// ---- VISUs/EtherCAT_Diag2.TcVIS
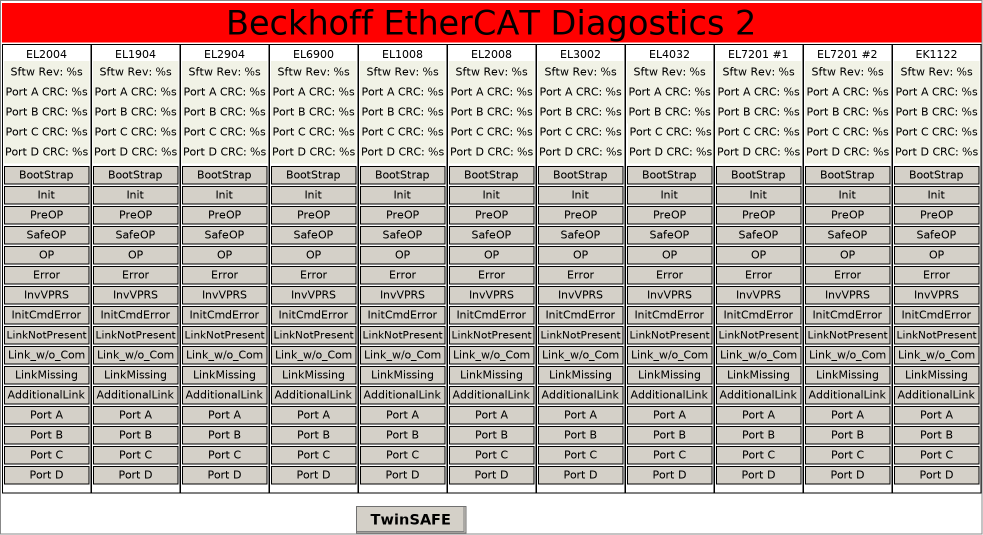
VISUALIZATION EtherCAT_Diag2  // 983x535
    Button (356,506 110x27), "TwinSAFE"
        OnMouseClick: change screen: TwinSAFE
    RoundedRectangle (2,3 979x39), "Beckhoff EtherCAT Diagostics 2"
    Group (2,42 89x451)
        RoundedRectangle (0,2 89x449)
        Label (2,0 85x25), "EL2004"
        Rectangle (2,19 85x22), "Sftw Rev: %s", text variable: g_iHMI_ProdCodeEL2004
        Rectangle (2,39 85x22), "Port A CRC: %s", text variable: g_stHMI_EL2004CrcErrorEx.portA
        Rectangle (2,59 85x22), "Port B CRC: %s", text variable: g_stHMI_EL2004CrcErrorEx.portB
        Rectangle (2,79 85x22), "Port C CRC: %s", text variable: g_stHMI_EL2004CrcErrorEx.portC
        Rectangle (2,99 85x22), "Port D CRC: %s", text variable: g_stHMI_EL2004CrcErrorEx.portD
        Rectangle (2,124 85x18), "BootStrap", colour toggle: g_stHMI_EL2004EcSlaveStateBits.bBootStrap
        Rectangle (2,144 85x18), "Init", colour toggle: g_stHMI_EL2004EcSlaveStateBits.bInit
        Rectangle (2,164 85x18), "PreOP", colour toggle: g_stHMI_EL2004EcSlaveStateBits.bPreop
        Rectangle (2,184 85x18), "SafeOP", colour toggle: g_stHMI_EL2004EcSlaveStateBits.bSafeOp
        Rectangle (2,204 85x18), "OP", colour toggle: g_stHMI_EL2004EcSlaveStateBits.bOp
        Rectangle (2,224 85x18), "Error", colour toggle: g_stHMI_EL2004EcSlaveStateBits.bError
        Rectangle (2,244 85x18), "InvVPRS", colour toggle: g_stHMI_EL2004EcSlaveStateBits.bInvVPRS
        Rectangle (2,264 85x18), "InitCmdError", colour toggle: g_stHMI_EL2004EcSlaveStateBits.bInitCmdError
        Rectangle (2,284 85x18), "LinkNotPresent", colour toggle: g_stHMI_EL2004EcSlaveStateBits.bLinkNotPresent
        Rectangle (2,304 85x18), "Link_w/o_Com", colour toggle: g_stHMI_EL2004EcSlaveStateBits.bLinkWithoutComm
        Rectangle (2,324 85x18), "LinkMissing", colour toggle: g_stHMI_EL2004EcSlaveStateBits.bLinkMissing
        Rectangle (2,344 85x18), "AdditionalLink", colour toggle: g_stHMI_EL2004EcSlaveStateBits.bAdditionalLink
        Rectangle (2,364 85x18), "Port A", colour toggle: g_stHMI_EL2004EcSlaveStateBits.bPortA
        Rectangle (2,384 85x18), "Port B", colour toggle: g_stHMI_EL2004EcSlaveStateBits.bPortB
        Rectangle (2,404 85x18), "Port C", colour toggle: g_stHMI_EL2004EcSlaveStateBits.bPortC
        Rectangle (2,424 85x18), "Port D", colour toggle: g_stHMI_EL2004EcSlaveStateBits.bPortD
    Group (91,42 89x451)
        RoundedRectangle (0,2 89x449)
        Label (2,0 85x25), "EL1904"
        Rectangle (2,19 85x22), "Sftw Rev: %s", text variable: g_iHMI_ProdCodeEL1904
        Rectangle (2,39 85x22), "Port A CRC: %s", text variable: g_stHMI_EL1904CrcErrorEx.portA
        Rectangle (2,59 85x22), "Port B CRC: %s", text variable: g_stHMI_EL1904CrcErrorEx.portB
        Rectangle (2,79 85x22), "Port C CRC: %s", text variable: g_stHMI_EL1904CrcErrorEx.portC
        Rectangle (2,99 85x22), "Port D CRC: %s", text variable: g_stHMI_EL1904CrcErrorEx.portD
        Rectangle (2,124 85x18), "BootStrap", colour toggle: g_stHMI_EL1904EcSlaveStateBits.bBootStrap
        Rectangle (2,144 85x18), "Init", colour toggle: g_stHMI_EL1904EcSlaveStateBits.bInit
        Rectangle (2,164 85x18), "PreOP", colour toggle: g_stHMI_EL1904EcSlaveStateBits.bPreop
        Rectangle (2,184 85x18), "SafeOP", colour toggle: g_stHMI_EL1904EcSlaveStateBits.bSafeOp
        Rectangle (2,204 85x18), "OP", colour toggle: g_stHMI_EL1904EcSlaveStateBits.bOp
        Rectangle (2,224 85x18), "Error", colour toggle: g_stHMI_EL1904EcSlaveStateBits.bError
        Rectangle (2,244 85x18), "InvVPRS", colour toggle: g_stHMI_EL1904EcSlaveStateBits.bInvVPRS
        Rectangle (2,264 85x18), "InitCmdError", colour toggle: g_stHMI_EL1904EcSlaveStateBits.bInitCmdError
        Rectangle (2,284 85x18), "LinkNotPresent", colour toggle: g_stHMI_EL1904EcSlaveStateBits.bLinkNotPresent
        Rectangle (2,304 85x18), "Link_w/o_Com", colour toggle: g_stHMI_EL1904EcSlaveStateBits.bLinkWithoutComm
        Rectangle (2,324 85x18), "LinkMissing", colour toggle: g_stHMI_EL1904EcSlaveStateBits.bLinkMissing
        Rectangle (2,344 85x18), "AdditionalLink", colour toggle: g_stHMI_EL1904EcSlaveStateBits.bAdditionalLink
        Rectangle (2,364 85x18), "Port A", colour toggle: g_stHMI_EL1904EcSlaveStateBits.bPortA
        Rectangle (2,384 85x18), "Port B", colour toggle: g_stHMI_EL1904EcSlaveStateBits.bPortB
        Rectangle (2,404 85x18), "Port C", colour toggle: g_stHMI_EL1904EcSlaveStateBits.bPortC
        Rectangle (2,424 85x18), "Port D", colour toggle: g_stHMI_EL1904EcSlaveStateBits.bPortD
    Group (180,42 89x451)
        RoundedRectangle (0,2 89x449)
        Label (2,0 85x25), "EL2904"
        Rectangle (2,19 85x22), "Sftw Rev: %s", text variable: g_iHMI_ProdCodeEL2904
        Rectangle (2,39 85x22), "Port A CRC: %s", text variable: g_stHMI_EL2904CrcErrorEx.portA
        Rectangle (2,59 85x22), "Port B CRC: %s", text variable: g_stHMI_EL2904CrcErrorEx.portB
        Rectangle (2,79 85x22), "Port C CRC: %s", text variable: g_stHMI_EL2904CrcErrorEx.portC
        Rectangle (2,99 85x22), "Port D CRC: %s", text variable: g_stHMI_EL2904CrcErrorEx.portD
        Rectangle (2,124 85x18), "BootStrap", colour toggle: g_stHMI_EL2904EcSlaveStateBits.bBootStrap
        Rectangle (2,144 85x18), "Init", colour toggle: g_stHMI_EL2904EcSlaveStateBits.bInit
        Rectangle (2,164 85x18), "PreOP", colour toggle: g_stHMI_EL2904EcSlaveStateBits.bPreop
        Rectangle (2,184 85x18), "SafeOP", colour toggle: g_stHMI_EL2904EcSlaveStateBits.bSafeOp
        Rectangle (2,204 85x18), "OP", colour toggle: g_stHMI_EL2904EcSlaveStateBits.bOp
        Rectangle (2,224 85x18), "Error", colour toggle: g_stHMI_EL2904EcSlaveStateBits.bError
        Rectangle (2,244 85x18), "InvVPRS", colour toggle: g_stHMI_EL2904EcSlaveStateBits.bInvVPRS
        Rectangle (2,264 85x18), "InitCmdError", colour toggle: g_stHMI_EL2904EcSlaveStateBits.bInitCmdError
        Rectangle (2,284 85x18), "LinkNotPresent", colour toggle: g_stHMI_EL2904EcSlaveStateBits.bLinkNotPresent
        Rectangle (2,304 85x18), "Link_w/o_Com", colour toggle: g_stHMI_EL2904EcSlaveStateBits.bLinkWithoutComm
        Rectangle (2,324 85x18), "LinkMissing", colour toggle: g_stHMI_EL2904EcSlaveStateBits.bLinkMissing
        Rectangle (2,344 85x18), "AdditionalLink", colour toggle: g_stHMI_EL2904EcSlaveStateBits.bAdditionalLink
        Rectangle (2,364 85x18), "Port A", colour toggle: g_stHMI_EL2904EcSlaveStateBits.bPortA
        Rectangle (2,384 85x18), "Port B", colour toggle: g_stHMI_EL2904EcSlaveStateBits.bPortB
        Rectangle (2,404 85x18), "Port C", colour toggle: g_stHMI_EL2904EcSlaveStateBits.bPortC
        Rectangle (2,424 85x18), "Port D", colour toggle: g_stHMI_EL2904EcSlaveStateBits.bPortD
    Group (269,42 89x451)
        RoundedRectangle (0,2 89x449)
        Label (2,0 85x25), "EL6900"
        Rectangle (2,19 85x22), "Sftw Rev: %s", text variable: g_iHMI_ProdCodeEL6900
        Rectangle (2,39 85x22), "Port A CRC: %s", text variable: g_stHMI_EL6900CrcErrorEx.portA
        Rectangle (2,59 85x22), "Port B CRC: %s", text variable: g_stHMI_EL6900CrcErrorEx.portB
        Rectangle (2,79 85x22), "Port C CRC: %s", text variable: g_stHMI_EL6900CrcErrorEx.portC
        Rectangle (2,99 85x22), "Port D CRC: %s", text variable: g_stHMI_EL6900CrcErrorEx.portD
        Rectangle (2,124 85x18), "BootStrap", colour toggle: g_stHMI_EL6900EcSlaveStateBits.bBootStrap
        Rectangle (2,144 85x18), "Init", colour toggle: g_stHMI_EL6900EcSlaveStateBits.bInit
        Rectangle (2,164 85x18), "PreOP", colour toggle: g_stHMI_EL6900EcSlaveStateBits.bPreop
        Rectangle (2,184 85x18), "SafeOP", colour toggle: g_stHMI_EL6900EcSlaveStateBits.bSafeOp
        Rectangle (2,204 85x18), "OP", colour toggle: g_stHMI_EL6900EcSlaveStateBits.bOp
        Rectangle (2,224 85x18), "Error", colour toggle: g_stHMI_EL6900EcSlaveStateBits.bError
        Rectangle (2,244 85x18), "InvVPRS", colour toggle: g_stHMI_EL6900EcSlaveStateBits.bInvVPRS
        Rectangle (2,264 85x18), "InitCmdError", colour toggle: g_stHMI_EL6900EcSlaveStateBits.bInitCmdError
        Rectangle (2,284 85x18), "LinkNotPresent", colour toggle: g_stHMI_EL6900EcSlaveStateBits.bLinkNotPresent
        Rectangle (2,304 85x18), "Link_w/o_Com", colour toggle: g_stHMI_EL6900EcSlaveStateBits.bLinkWithoutComm
        Rectangle (2,324 85x18), "LinkMissing", colour toggle: g_stHMI_EL6900EcSlaveStateBits.bLinkMissing
        Rectangle (2,344 85x18), "AdditionalLink", colour toggle: g_stHMI_EL6900EcSlaveStateBits.bAdditionalLink
        Rectangle (2,364 85x18), "Port A", colour toggle: g_stHMI_EL6900EcSlaveStateBits.bPortA
        Rectangle (2,384 85x18), "Port B", colour toggle: g_stHMI_EL6900EcSlaveStateBits.bPortB
        Rectangle (2,404 85x18), "Port C", colour toggle: g_stHMI_EL6900EcSlaveStateBits.bPortC
        Rectangle (2,424 85x18), "Port D", colour toggle: g_stHMI_EL6900EcSlaveStateBits.bPortD
    Group (358,42 89x451)
        RoundedRectangle (0,2 89x449)
        Label (2,0 85x25), "EL1008"
        Rectangle (2,19 85x22), "Sftw Rev: %s", text variable: g_iHMI_ProdCodeEL1008
        Rectangle (2,39 85x22), "Port A CRC: %s", text variable: g_stHMI_EL1008CrcErrorEx.portA
        Rectangle (2,59 85x22), "Port B CRC: %s", text variable: g_stHMI_EL1008CrcErrorEx.portB
        Rectangle (2,79 85x22), "Port C CRC: %s", text variable: g_stHMI_EL1008CrcErrorEx.portC
        Rectangle (2,99 85x22), "Port D CRC: %s", text variable: g_stHMI_EL1008CrcErrorEx.portD
        Rectangle (2,124 85x18), "BootStrap", colour toggle: g_stHMI_EL1008EcSlaveStateBits.bBootStrap
        Rectangle (2,144 85x18), "Init", colour toggle: g_stHMI_EL1008EcSlaveStateBits.bInit
        Rectangle (2,164 85x18), "PreOP", colour toggle: g_stHMI_EL1008EcSlaveStateBits.bPreop
        Rectangle (2,184 85x18), "SafeOP", colour toggle: g_stHMI_EL1008EcSlaveStateBits.bSafeOp
        Rectangle (2,204 85x18), "OP", colour toggle: g_stHMI_EL1008EcSlaveStateBits.bOp
        Rectangle (2,224 85x18), "Error", colour toggle: g_stHMI_EL1008EcSlaveStateBits.bError
        Rectangle (2,244 85x18), "InvVPRS", colour toggle: g_stHMI_EL1008EcSlaveStateBits.bInvVPRS
        Rectangle (2,264 85x18), "InitCmdError", colour toggle: g_stHMI_EL1008EcSlaveStateBits.bInitCmdError
        Rectangle (2,284 85x18), "LinkNotPresent", colour toggle: g_stHMI_EL1008EcSlaveStateBits.bLinkNotPresent
        Rectangle (2,304 85x18), "Link_w/o_Com", colour toggle: g_stHMI_EL1008EcSlaveStateBits.bLinkWithoutComm
        Rectangle (2,324 85x18), "LinkMissing", colour toggle: g_stHMI_EL1008EcSlaveStateBits.bLinkMissing
        Rectangle (2,344 85x18), "AdditionalLink", colour toggle: g_stHMI_EL1008EcSlaveStateBits.bAdditionalLink
        Rectangle (2,364 85x18), "Port A", colour toggle: g_stHMI_EL1008EcSlaveStateBits.bPortA
        Rectangle (2,384 85x18), "Port B", colour toggle: g_stHMI_EL1008EcSlaveStateBits.bPortB
        Rectangle (2,404 85x18), "Port C", colour toggle: g_stHMI_EL1008EcSlaveStateBits.bPortC
        Rectangle (2,424 85x18), "Port D", colour toggle: g_stHMI_EL1008EcSlaveStateBits.bPortD
    Group (447,42 89x451)
        RoundedRectangle (0,2 89x449)
        Label (2,0 85x25), "EL2008"
        Rectangle (2,19 85x22), "Sftw Rev: %s", text variable: g_iHMI_ProdCodeEL2008
        Rectangle (2,39 85x22), "Port A CRC: %s", text variable: g_stHMI_EL2008CrcErrorEx.portA
        Rectangle (2,59 85x22), "Port B CRC: %s", text variable: g_stHMI_EL2008CrcErrorEx.portB
        Rectangle (2,79 85x22), "Port C CRC: %s", text variable: g_stHMI_EL2008CrcErrorEx.portC
        Rectangle (2,99 85x22), "Port D CRC: %s", text variable: g_stHMI_EL2008CrcErrorEx.portD
        Rectangle (2,124 85x18), "BootStrap", colour toggle: g_stHMI_EL2008EcSlaveStateBits.bBootStrap
        Rectangle (2,144 85x18), "Init", colour toggle: g_stHMI_EL2008EcSlaveStateBits.bInit
        Rectangle (2,164 85x18), "PreOP", colour toggle: g_stHMI_EL2008EcSlaveStateBits.bPreop
        Rectangle (2,184 85x18), "SafeOP", colour toggle: g_stHMI_EL2008EcSlaveStateBits.bSafeOp
        Rectangle (2,204 85x18), "OP", colour toggle: g_stHMI_EL2008EcSlaveStateBits.bOp
        Rectangle (2,224 85x18), "Error", colour toggle: g_stHMI_EL2008EcSlaveStateBits.bError
        Rectangle (2,244 85x18), "InvVPRS", colour toggle: g_stHMI_EL2008EcSlaveStateBits.bInvVPRS
        Rectangle (2,264 85x18), "InitCmdError", colour toggle: g_stHMI_EL2008EcSlaveStateBits.bInitCmdError
        Rectangle (2,284 85x18), "LinkNotPresent", colour toggle: g_stHMI_EL2008EcSlaveStateBits.bLinkNotPresent
        Rectangle (2,304 85x18), "Link_w/o_Com", colour toggle: g_stHMI_EL2008EcSlaveStateBits.bLinkWithoutComm
        Rectangle (2,324 85x18), "LinkMissing", colour toggle: g_stHMI_EL2008EcSlaveStateBits.bLinkMissing
        Rectangle (2,344 85x18), "AdditionalLink", colour toggle: g_stHMI_EL2008EcSlaveStateBits.bAdditionalLink
        Rectangle (2,364 85x18), "Port A", colour toggle: g_stHMI_EL2008EcSlaveStateBits.bPortA
        Rectangle (2,384 85x18), "Port B", colour toggle: g_stHMI_EL2008EcSlaveStateBits.bPortB
        Rectangle (2,404 85x18), "Port C", colour toggle: g_stHMI_EL2008EcSlaveStateBits.bPortC
        Rectangle (2,424 85x18), "Port D", colour toggle: g_stHMI_EL2008EcSlaveStateBits.bPortD
    Group (536,42 89x451)
        RoundedRectangle (0,2 89x449)
        Label (2,0 85x25), "EL3002"
        Rectangle (2,19 85x22), "Sftw Rev: %s", text variable: g_iHMI_ProdCodeEL3002
        Rectangle (2,39 85x22), "Port A CRC: %s", text variable: g_stHMI_EL3002CrcErrorEx.portA
        Rectangle (2,59 85x22), "Port B CRC: %s", text variable: g_stHMI_EL3002CrcErrorEx.portB
        Rectangle (2,79 85x22), "Port C CRC: %s", text variable: g_stHMI_EL3002CrcErrorEx.portC
        Rectangle (2,99 85x22), "Port D CRC: %s", text variable: g_stHMI_EL3002CrcErrorEx.portD
        Rectangle (2,124 85x18), "BootStrap", colour toggle: g_stHMI_EL3002EcSlaveStateBits.bBootStrap
        Rectangle (2,144 85x18), "Init", colour toggle: g_stHMI_EL3002EcSlaveStateBits.bInit
        Rectangle (2,164 85x18), "PreOP", colour toggle: g_stHMI_EL3002EcSlaveStateBits.bPreop
        Rectangle (2,184 85x18), "SafeOP", colour toggle: g_stHMI_EL3002EcSlaveStateBits.bSafeOp
        Rectangle (2,204 85x18), "OP", colour toggle: g_stHMI_EL3002EcSlaveStateBits.bOp
        Rectangle (2,224 85x18), "Error", colour toggle: g_stHMI_EL3002EcSlaveStateBits.bError
        Rectangle (2,244 85x18), "InvVPRS", colour toggle: g_stHMI_EL3002EcSlaveStateBits.bInvVPRS
        Rectangle (2,264 85x18), "InitCmdError", colour toggle: g_stHMI_EL3002EcSlaveStateBits.bInitCmdError
        Rectangle (2,284 85x18), "LinkNotPresent", colour toggle: g_stHMI_EL3002EcSlaveStateBits.bLinkNotPresent
        Rectangle (2,304 85x18), "Link_w/o_Com", colour toggle: g_stHMI_EL3002EcSlaveStateBits.bLinkWithoutComm
        Rectangle (2,324 85x18), "LinkMissing", colour toggle: g_stHMI_EL3002EcSlaveStateBits.bLinkMissing
        Rectangle (2,344 85x18), "AdditionalLink", colour toggle: g_stHMI_EL3002EcSlaveStateBits.bAdditionalLink
        Rectangle (2,364 85x18), "Port A", colour toggle: g_stHMI_EL3002EcSlaveStateBits.bPortA
        Rectangle (2,384 85x18), "Port B", colour toggle: g_stHMI_EL3002EcSlaveStateBits.bPortB
        Rectangle (2,404 85x18), "Port C", colour toggle: g_stHMI_EL3002EcSlaveStateBits.bPortC
        Rectangle (2,424 85x18), "Port D", colour toggle: g_stHMI_EL3002EcSlaveStateBits.bPortD
    RoundedRectangle (625,44 89x449)
    Label (627,42 85x25), "EL4032"
    Rectangle (627,61 85x22), "Sftw Rev: %s", text variable: g_iHMI_ProdCodeEL4032
    Rectangle (627,81 85x22), "Port A CRC: %s", text variable: g_stHMI_EL4032CrcErrorEx.portA
    Rectangle (627,101 85x22), "Port B CRC: %s", text variable: g_stHMI_EL4032CrcErrorEx.portB
    Rectangle (628,121 85x22), "Port C CRC: %s", text variable: g_stHMI_EL4032CrcErrorEx.portC
    Rectangle (628,141 85x22), "Port D CRC: %s", text variable: g_stHMI_EL4032CrcErrorEx.portD
    Rectangle (627,166 85x18), "BootStrap", colour toggle: g_stHMI_EL4032EcSlaveStateBits.bBootStrap
    Rectangle (627,186 85x18), "Init", colour toggle: g_stHMI_EL4032EcSlaveStateBits.bInit
    Rectangle (627,206 85x18), "PreOP", colour toggle: g_stHMI_EL4032EcSlaveStateBits.bPreop
    Rectangle (627,226 85x18), "SafeOP", colour toggle: g_stHMI_EL4032EcSlaveStateBits.bSafeOp
    Rectangle (627,246 85x18), "OP", colour toggle: g_stHMI_EL4032EcSlaveStateBits.bOp
    Rectangle (627,266 85x18), "Error", colour toggle: g_stHMI_EL4032EcSlaveStateBits.bError
    Rectangle (627,286 85x18), "InvVPRS", colour toggle: g_stHMI_EL4032EcSlaveStateBits.bInvVPRS
    Rectangle (627,306 85x18), "InitCmdError", colour toggle: g_stHMI_EL4032EcSlaveStateBits.bInitCmdError
    Rectangle (627,326 85x18), "LinkNotPresent", colour toggle: g_stHMI_EL4032EcSlaveStateBits.bLinkNotPresent
    Rectangle (627,346 85x18), "Link_w/o_Com", colour toggle: g_stHMI_EL4032EcSlaveStateBits.bLinkWithoutComm
    Rectangle (627,366 85x18), "LinkMissing", colour toggle: g_stHMI_EL4032EcSlaveStateBits.bLinkMissing
    Rectangle (627,386 85x18), "AdditionalLink", colour toggle: g_stHMI_EL4032EcSlaveStateBits.bAdditionalLink
    Rectangle (627,406 85x18), "Port A", colour toggle: g_stHMI_EL4032EcSlaveStateBits.bPortA
    Rectangle (627,426 85x18), "Port B", colour toggle: g_stHMI_EL4032EcSlaveStateBits.bPortB
    Rectangle (627,446 85x18), "Port C", colour toggle: g_stHMI_EL4032EcSlaveStateBits.bPortC
    Rectangle (627,466 85x18), "Port D", colour toggle: g_stHMI_EL4032EcSlaveStateBits.bPortD
    Group (714,42 89x451)
        RoundedRectangle (0,2 89x449)
        Label (2,0 85x25), "EL7201 #1"
        Rectangle (2,19 85x22), "Sftw Rev: %s", text variable: g_iHMI_ProdCodeEL7201_1
        Rectangle (2,39 85x22), "Port A CRC: %s", text variable: g_stHMI_EL7201_1CrcErrorEx.portA
        Rectangle (2,59 85x22), "Port B CRC: %s", text variable: g_stHMI_EL7201_1CrcErrorEx.portB
        Rectangle (2,79 85x22), "Port C CRC: %s", text variable: g_stHMI_EL7201_1CrcErrorEx.portC
        Rectangle (2,99 85x22), "Port D CRC: %s", text variable: g_stHMI_EL7201_1CrcErrorEx.portD
        Rectangle (2,124 85x18), "BootStrap", colour toggle: g_stHMI_EL7201_1EcSlaveStateBits.bBootStrap
        Rectangle (2,144 85x18), "Init", colour toggle: g_stHMI_EL7201_1EcSlaveStateBits.bInit
        Rectangle (2,164 85x18), "PreOP", colour toggle: g_stHMI_EL7201_1EcSlaveStateBits.bPreop
        Rectangle (2,184 85x18), "SafeOP", colour toggle: g_stHMI_EL7201_1EcSlaveStateBits.bSafeOp
        Rectangle (2,204 85x18), "OP", colour toggle: g_stHMI_EL7201_1EcSlaveStateBits.bOp
        Rectangle (2,224 85x18), "Error", colour toggle: g_stHMI_EL7201_1EcSlaveStateBits.bError
        Rectangle (2,244 85x18), "InvVPRS", colour toggle: g_stHMI_EL7201_1EcSlaveStateBits.bInvVPRS
        Rectangle (2,264 85x18), "InitCmdError", colour toggle: g_stHMI_EL7201_1EcSlaveStateBits.bInitCmdError
        Rectangle (2,284 85x18), "LinkNotPresent", colour toggle: g_stHMI_EL7201_1EcSlaveStateBits.bLinkNotPresent
        Rectangle (2,304 85x18), "Link_w/o_Com", colour toggle: g_stHMI_EL7201_1EcSlaveStateBits.bLinkWithoutComm
        Rectangle (2,324 85x18), "LinkMissing", colour toggle: g_stHMI_EL7201_1EcSlaveStateBits.bLinkMissing
        Rectangle (2,344 85x18), "AdditionalLink", colour toggle: g_stHMI_EL7201_1EcSlaveStateBits.bAdditionalLink
        Rectangle (2,364 85x18), "Port A", colour toggle: g_stHMI_EL7201_1EcSlaveStateBits.bPortA
        Rectangle (2,384 85x18), "Port B", colour toggle: g_stHMI_EL7201_1EcSlaveStateBits.bPortB
        Rectangle (2,404 85x18), "Port C", colour toggle: g_stHMI_EL7201_1EcSlaveStateBits.bPortC
        Rectangle (2,424 85x18), "Port D", colour toggle: g_stHMI_EL7201_1EcSlaveStateBits.bPortD
    Group (803,42 89x451)
        RoundedRectangle (0,2 89x449)
        Label (2,0 85x25), "EL7201 #2"
        Rectangle (2,19 85x22), "Sftw Rev: %s", text variable: g_iHMI_ProdCodeEL7201_2
        Rectangle (2,39 85x22), "Port A CRC: %s", text variable: g_stHMI_EL7201_2CrcErrorEx.portA
        Rectangle (2,59 85x22), "Port B CRC: %s", text variable: g_stHMI_EL7201_2CrcErrorEx.portB
        Rectangle (2,79 85x22), "Port C CRC: %s", text variable: g_stHMI_EL7201_2CrcErrorEx.portC
        Rectangle (2,99 85x22), "Port D CRC: %s", text variable: g_stHMI_EL7201_2CrcErrorEx.portD
        Rectangle (2,124 85x18), "BootStrap", colour toggle: g_stHMI_EL7201_2EcSlaveStateBits.bBootStrap
        Rectangle (2,144 85x18), "Init", colour toggle: g_stHMI_EL7201_2EcSlaveStateBits.bInit
        Rectangle (2,164 85x18), "PreOP", colour toggle: g_stHMI_EL7201_2EcSlaveStateBits.bPreop
        Rectangle (2,184 85x18), "SafeOP", colour toggle: g_stHMI_EL7201_2EcSlaveStateBits.bSafeOp
        Rectangle (2,204 85x18), "OP", colour toggle: g_stHMI_EL7201_2EcSlaveStateBits.bOp
        Rectangle (2,224 85x18), "Error", colour toggle: g_stHMI_EL7201_2EcSlaveStateBits.bError
        Rectangle (2,244 85x18), "InvVPRS", colour toggle: g_stHMI_EL7201_2EcSlaveStateBits.bInvVPRS
        Rectangle (2,264 85x18), "InitCmdError", colour toggle: g_stHMI_EL7201_2EcSlaveStateBits.bInitCmdError
        Rectangle (2,284 85x18), "LinkNotPresent", colour toggle: g_stHMI_EL7201_2EcSlaveStateBits.bLinkNotPresent
        Rectangle (2,304 85x18), "Link_w/o_Com", colour toggle: g_stHMI_EL7201_2EcSlaveStateBits.bLinkWithoutComm
        Rectangle (2,324 85x18), "LinkMissing", colour toggle: g_stHMI_EL7201_2EcSlaveStateBits.bLinkMissing
        Rectangle (2,344 85x18), "AdditionalLink", colour toggle: g_stHMI_EL7201_2EcSlaveStateBits.bAdditionalLink
        Rectangle (2,364 85x18), "Port A", colour toggle: g_stHMI_EL7201_2EcSlaveStateBits.bPortA
        Rectangle (2,384 85x18), "Port B", colour toggle: g_stHMI_EL7201_2EcSlaveStateBits.bPortB
        Rectangle (2,404 85x18), "Port C", colour toggle: g_stHMI_EL7201_2EcSlaveStateBits.bPortC
        Rectangle (2,424 85x18), "Port D", colour toggle: g_stHMI_EL7201_2EcSlaveStateBits.bPortD
    Group (892,42 89x451)
        RoundedRectangle (0,2 89x449)
        Label (2,0 85x25), "EK1122"
        Rectangle (2,19 85x22), "Sftw Rev: %s", text variable: g_iHMI_ProdCodeEK1122
        Rectangle (2,39 85x22), "Port A CRC: %s", text variable: g_stHMI_EK1122_CrcErrorEx.portA
        Rectangle (2,59 85x22), "Port B CRC: %s", text variable: g_stHMI_EK1122_CrcErrorEx.portB
        Rectangle (2,79 85x22), "Port C CRC: %s", text variable: g_stHMI_EK1122_CrcErrorEx.portC
        Rectangle (2,99 85x22), "Port D CRC: %s", text variable: g_stHMI_EK1122_CrcErrorEx.portD
        Rectangle (2,124 85x18), "BootStrap", colour toggle: g_stHMI_EK1122_EcSlaveStateBits.bBootStrap
        Rectangle (2,144 85x18), "Init", colour toggle: g_stHMI_EK1122_EcSlaveStateBits.bInit
        Rectangle (2,164 85x18), "PreOP", colour toggle: g_stHMI_EK1122_EcSlaveStateBits.bPreop
        Rectangle (2,184 85x18), "SafeOP", colour toggle: g_stHMI_EK1122_EcSlaveStateBits.bSafeOp
        Rectangle (2,204 85x18), "OP", colour toggle: g_stHMI_EK1122_EcSlaveStateBits.bOp
        Rectangle (2,224 85x18), "Error", colour toggle: g_stHMI_EK1122_EcSlaveStateBits.bError
        Rectangle (2,244 85x18), "InvVPRS", colour toggle: g_stHMI_EK1122_EcSlaveStateBits.bInvVPRS
        Rectangle (2,264 85x18), "InitCmdError", colour toggle: g_stHMI_EK1122_EcSlaveStateBits.bInitCmdError
        Rectangle (2,284 85x18), "LinkNotPresent", colour toggle: g_stHMI_EK1122_EcSlaveStateBits.bLinkNotPresent
        Rectangle (2,304 85x18), "Link_w/o_Com", colour toggle: g_stHMI_EK1122_EcSlaveStateBits.bLinkWithoutComm
        Rectangle (2,324 85x18), "LinkMissing", colour toggle: g_stHMI_EK1122_EcSlaveStateBits.bLinkMissing
        Rectangle (2,344 85x18), "AdditionalLink", colour toggle: g_stHMI_EK1122_EcSlaveStateBits.bAdditionalLink
        Rectangle (2,364 85x18), "Port A", colour toggle: g_stHMI_EK1122_EcSlaveStateBits.bPortA
        Rectangle (2,384 85x18), "Port B", colour toggle: g_stHMI_EK1122_EcSlaveStateBits.bPortB
        Rectangle (2,404 85x18), "Port C", colour toggle: g_stHMI_EK1122_EcSlaveStateBits.bPortC
        Rectangle (2,424 85x18), "Port D", colour toggle: g_stHMI_EK1122_EcSlaveStateBits.bPortD
END_VISUALIZATION

// ---- VISUs/EtherCAT_Diag2.TcVIS
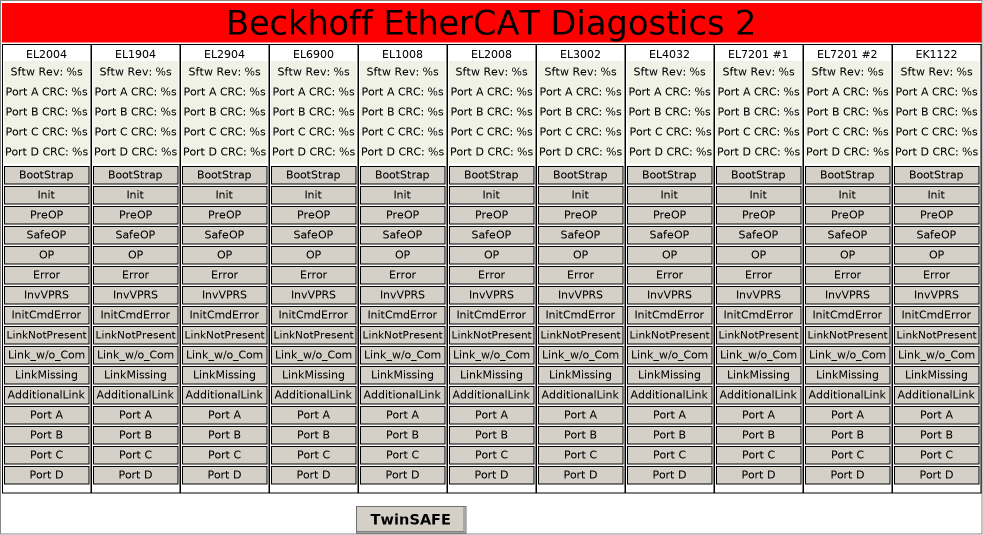
VISUALIZATION EtherCAT_Diag2  // 983x535
    Button (356,506 110x27), "TwinSAFE"
        OnMouseClick: change screen: TwinSAFE
    RoundedRectangle (2,3 979x39), "Beckhoff EtherCAT Diagostics 2"
    Group (2,42 89x451)
        RoundedRectangle (0,2 89x449)
        Label (2,0 85x25), "EL2004"
        Rectangle (2,19 85x22), "Sftw Rev: %s", text variable: g_iHMI_ProdCodeEL2004
        Rectangle (2,39 85x22), "Port A CRC: %s", text variable: g_stHMI_EL2004CrcErrorEx.portA
        Rectangle (2,59 85x22), "Port B CRC: %s", text variable: g_stHMI_EL2004CrcErrorEx.portB
        Rectangle (2,79 85x22), "Port C CRC: %s", text variable: g_stHMI_EL2004CrcErrorEx.portC
        Rectangle (2,99 85x22), "Port D CRC: %s", text variable: g_stHMI_EL2004CrcErrorEx.portD
        Rectangle (2,124 85x18), "BootStrap", colour toggle: g_stHMI_EL2004EcSlaveStateBits.bBootStrap
        Rectangle (2,144 85x18), "Init", colour toggle: g_stHMI_EL2004EcSlaveStateBits.bInit
        Rectangle (2,164 85x18), "PreOP", colour toggle: g_stHMI_EL2004EcSlaveStateBits.bPreop
        Rectangle (2,184 85x18), "SafeOP", colour toggle: g_stHMI_EL2004EcSlaveStateBits.bSafeOp
        Rectangle (2,204 85x18), "OP", colour toggle: g_stHMI_EL2004EcSlaveStateBits.bOp
        Rectangle (2,224 85x18), "Error", colour toggle: g_stHMI_EL2004EcSlaveStateBits.bError
        Rectangle (2,244 85x18), "InvVPRS", colour toggle: g_stHMI_EL2004EcSlaveStateBits.bInvVPRS
        Rectangle (2,264 85x18), "InitCmdError", colour toggle: g_stHMI_EL2004EcSlaveStateBits.bInitCmdError
        Rectangle (2,284 85x18), "LinkNotPresent", colour toggle: g_stHMI_EL2004EcSlaveStateBits.bLinkNotPresent
        Rectangle (2,304 85x18), "Link_w/o_Com", colour toggle: g_stHMI_EL2004EcSlaveStateBits.bLinkWithoutComm
        Rectangle (2,324 85x18), "LinkMissing", colour toggle: g_stHMI_EL2004EcSlaveStateBits.bLinkMissing
        Rectangle (2,344 85x18), "AdditionalLink", colour toggle: g_stHMI_EL2004EcSlaveStateBits.bAdditionalLink
        Rectangle (2,364 85x18), "Port A", colour toggle: g_stHMI_EL2004EcSlaveStateBits.bPortA
        Rectangle (2,384 85x18), "Port B", colour toggle: g_stHMI_EL2004EcSlaveStateBits.bPortB
        Rectangle (2,404 85x18), "Port C", colour toggle: g_stHMI_EL2004EcSlaveStateBits.bPortC
        Rectangle (2,424 85x18), "Port D", colour toggle: g_stHMI_EL2004EcSlaveStateBits.bPortD
    Group (91,42 89x451)
        RoundedRectangle (0,2 89x449)
        Label (2,0 85x25), "EL1904"
        Rectangle (2,19 85x22), "Sftw Rev: %s", text variable: g_iHMI_ProdCodeEL1904
        Rectangle (2,39 85x22), "Port A CRC: %s", text variable: g_stHMI_EL1904CrcErrorEx.portA
        Rectangle (2,59 85x22), "Port B CRC: %s", text variable: g_stHMI_EL1904CrcErrorEx.portB
        Rectangle (2,79 85x22), "Port C CRC: %s", text variable: g_stHMI_EL1904CrcErrorEx.portC
        Rectangle (2,99 85x22), "Port D CRC: %s", text variable: g_stHMI_EL1904CrcErrorEx.portD
        Rectangle (2,124 85x18), "BootStrap", colour toggle: g_stHMI_EL1904EcSlaveStateBits.bBootStrap
        Rectangle (2,144 85x18), "Init", colour toggle: g_stHMI_EL1904EcSlaveStateBits.bInit
        Rectangle (2,164 85x18), "PreOP", colour toggle: g_stHMI_EL1904EcSlaveStateBits.bPreop
        Rectangle (2,184 85x18), "SafeOP", colour toggle: g_stHMI_EL1904EcSlaveStateBits.bSafeOp
        Rectangle (2,204 85x18), "OP", colour toggle: g_stHMI_EL1904EcSlaveStateBits.bOp
        Rectangle (2,224 85x18), "Error", colour toggle: g_stHMI_EL1904EcSlaveStateBits.bError
        Rectangle (2,244 85x18), "InvVPRS", colour toggle: g_stHMI_EL1904EcSlaveStateBits.bInvVPRS
        Rectangle (2,264 85x18), "InitCmdError", colour toggle: g_stHMI_EL1904EcSlaveStateBits.bInitCmdError
        Rectangle (2,284 85x18), "LinkNotPresent", colour toggle: g_stHMI_EL1904EcSlaveStateBits.bLinkNotPresent
        Rectangle (2,304 85x18), "Link_w/o_Com", colour toggle: g_stHMI_EL1904EcSlaveStateBits.bLinkWithoutComm
        Rectangle (2,324 85x18), "LinkMissing", colour toggle: g_stHMI_EL1904EcSlaveStateBits.bLinkMissing
        Rectangle (2,344 85x18), "AdditionalLink", colour toggle: g_stHMI_EL1904EcSlaveStateBits.bAdditionalLink
        Rectangle (2,364 85x18), "Port A", colour toggle: g_stHMI_EL1904EcSlaveStateBits.bPortA
        Rectangle (2,384 85x18), "Port B", colour toggle: g_stHMI_EL1904EcSlaveStateBits.bPortB
        Rectangle (2,404 85x18), "Port C", colour toggle: g_stHMI_EL1904EcSlaveStateBits.bPortC
        Rectangle (2,424 85x18), "Port D", colour toggle: g_stHMI_EL1904EcSlaveStateBits.bPortD
    Group (180,42 89x451)
        RoundedRectangle (0,2 89x449)
        Label (2,0 85x25), "EL2904"
        Rectangle (2,19 85x22), "Sftw Rev: %s", text variable: g_iHMI_ProdCodeEL2904
        Rectangle (2,39 85x22), "Port A CRC: %s", text variable: g_stHMI_EL2904CrcErrorEx.portA
        Rectangle (2,59 85x22), "Port B CRC: %s", text variable: g_stHMI_EL2904CrcErrorEx.portB
        Rectangle (2,79 85x22), "Port C CRC: %s", text variable: g_stHMI_EL2904CrcErrorEx.portC
        Rectangle (2,99 85x22), "Port D CRC: %s", text variable: g_stHMI_EL2904CrcErrorEx.portD
        Rectangle (2,124 85x18), "BootStrap", colour toggle: g_stHMI_EL2904EcSlaveStateBits.bBootStrap
        Rectangle (2,144 85x18), "Init", colour toggle: g_stHMI_EL2904EcSlaveStateBits.bInit
        Rectangle (2,164 85x18), "PreOP", colour toggle: g_stHMI_EL2904EcSlaveStateBits.bPreop
        Rectangle (2,184 85x18), "SafeOP", colour toggle: g_stHMI_EL2904EcSlaveStateBits.bSafeOp
        Rectangle (2,204 85x18), "OP", colour toggle: g_stHMI_EL2904EcSlaveStateBits.bOp
        Rectangle (2,224 85x18), "Error", colour toggle: g_stHMI_EL2904EcSlaveStateBits.bError
        Rectangle (2,244 85x18), "InvVPRS", colour toggle: g_stHMI_EL2904EcSlaveStateBits.bInvVPRS
        Rectangle (2,264 85x18), "InitCmdError", colour toggle: g_stHMI_EL2904EcSlaveStateBits.bInitCmdError
        Rectangle (2,284 85x18), "LinkNotPresent", colour toggle: g_stHMI_EL2904EcSlaveStateBits.bLinkNotPresent
        Rectangle (2,304 85x18), "Link_w/o_Com", colour toggle: g_stHMI_EL2904EcSlaveStateBits.bLinkWithoutComm
        Rectangle (2,324 85x18), "LinkMissing", colour toggle: g_stHMI_EL2904EcSlaveStateBits.bLinkMissing
        Rectangle (2,344 85x18), "AdditionalLink", colour toggle: g_stHMI_EL2904EcSlaveStateBits.bAdditionalLink
        Rectangle (2,364 85x18), "Port A", colour toggle: g_stHMI_EL2904EcSlaveStateBits.bPortA
        Rectangle (2,384 85x18), "Port B", colour toggle: g_stHMI_EL2904EcSlaveStateBits.bPortB
        Rectangle (2,404 85x18), "Port C", colour toggle: g_stHMI_EL2904EcSlaveStateBits.bPortC
        Rectangle (2,424 85x18), "Port D", colour toggle: g_stHMI_EL2904EcSlaveStateBits.bPortD
    Group (269,42 89x451)
        RoundedRectangle (0,2 89x449)
        Label (2,0 85x25), "EL6900"
        Rectangle (2,19 85x22), "Sftw Rev: %s", text variable: g_iHMI_ProdCodeEL6900
        Rectangle (2,39 85x22), "Port A CRC: %s", text variable: g_stHMI_EL6900CrcErrorEx.portA
        Rectangle (2,59 85x22), "Port B CRC: %s", text variable: g_stHMI_EL6900CrcErrorEx.portB
        Rectangle (2,79 85x22), "Port C CRC: %s", text variable: g_stHMI_EL6900CrcErrorEx.portC
        Rectangle (2,99 85x22), "Port D CRC: %s", text variable: g_stHMI_EL6900CrcErrorEx.portD
        Rectangle (2,124 85x18), "BootStrap", colour toggle: g_stHMI_EL6900EcSlaveStateBits.bBootStrap
        Rectangle (2,144 85x18), "Init", colour toggle: g_stHMI_EL6900EcSlaveStateBits.bInit
        Rectangle (2,164 85x18), "PreOP", colour toggle: g_stHMI_EL6900EcSlaveStateBits.bPreop
        Rectangle (2,184 85x18), "SafeOP", colour toggle: g_stHMI_EL6900EcSlaveStateBits.bSafeOp
        Rectangle (2,204 85x18), "OP", colour toggle: g_stHMI_EL6900EcSlaveStateBits.bOp
        Rectangle (2,224 85x18), "Error", colour toggle: g_stHMI_EL6900EcSlaveStateBits.bError
        Rectangle (2,244 85x18), "InvVPRS", colour toggle: g_stHMI_EL6900EcSlaveStateBits.bInvVPRS
        Rectangle (2,264 85x18), "InitCmdError", colour toggle: g_stHMI_EL6900EcSlaveStateBits.bInitCmdError
        Rectangle (2,284 85x18), "LinkNotPresent", colour toggle: g_stHMI_EL6900EcSlaveStateBits.bLinkNotPresent
        Rectangle (2,304 85x18), "Link_w/o_Com", colour toggle: g_stHMI_EL6900EcSlaveStateBits.bLinkWithoutComm
        Rectangle (2,324 85x18), "LinkMissing", colour toggle: g_stHMI_EL6900EcSlaveStateBits.bLinkMissing
        Rectangle (2,344 85x18), "AdditionalLink", colour toggle: g_stHMI_EL6900EcSlaveStateBits.bAdditionalLink
        Rectangle (2,364 85x18), "Port A", colour toggle: g_stHMI_EL6900EcSlaveStateBits.bPortA
        Rectangle (2,384 85x18), "Port B", colour toggle: g_stHMI_EL6900EcSlaveStateBits.bPortB
        Rectangle (2,404 85x18), "Port C", colour toggle: g_stHMI_EL6900EcSlaveStateBits.bPortC
        Rectangle (2,424 85x18), "Port D", colour toggle: g_stHMI_EL6900EcSlaveStateBits.bPortD
    Group (358,42 89x451)
        RoundedRectangle (0,2 89x449)
        Label (2,0 85x25), "EL1008"
        Rectangle (2,19 85x22), "Sftw Rev: %s", text variable: g_iHMI_ProdCodeEL1008
        Rectangle (2,39 85x22), "Port A CRC: %s", text variable: g_stHMI_EL1008CrcErrorEx.portA
        Rectangle (2,59 85x22), "Port B CRC: %s", text variable: g_stHMI_EL1008CrcErrorEx.portB
        Rectangle (2,79 85x22), "Port C CRC: %s", text variable: g_stHMI_EL1008CrcErrorEx.portC
        Rectangle (2,99 85x22), "Port D CRC: %s", text variable: g_stHMI_EL1008CrcErrorEx.portD
        Rectangle (2,124 85x18), "BootStrap", colour toggle: g_stHMI_EL1008EcSlaveStateBits.bBootStrap
        Rectangle (2,144 85x18), "Init", colour toggle: g_stHMI_EL1008EcSlaveStateBits.bInit
        Rectangle (2,164 85x18), "PreOP", colour toggle: g_stHMI_EL1008EcSlaveStateBits.bPreop
        Rectangle (2,184 85x18), "SafeOP", colour toggle: g_stHMI_EL1008EcSlaveStateBits.bSafeOp
        Rectangle (2,204 85x18), "OP", colour toggle: g_stHMI_EL1008EcSlaveStateBits.bOp
        Rectangle (2,224 85x18), "Error", colour toggle: g_stHMI_EL1008EcSlaveStateBits.bError
        Rectangle (2,244 85x18), "InvVPRS", colour toggle: g_stHMI_EL1008EcSlaveStateBits.bInvVPRS
        Rectangle (2,264 85x18), "InitCmdError", colour toggle: g_stHMI_EL1008EcSlaveStateBits.bInitCmdError
        Rectangle (2,284 85x18), "LinkNotPresent", colour toggle: g_stHMI_EL1008EcSlaveStateBits.bLinkNotPresent
        Rectangle (2,304 85x18), "Link_w/o_Com", colour toggle: g_stHMI_EL1008EcSlaveStateBits.bLinkWithoutComm
        Rectangle (2,324 85x18), "LinkMissing", colour toggle: g_stHMI_EL1008EcSlaveStateBits.bLinkMissing
        Rectangle (2,344 85x18), "AdditionalLink", colour toggle: g_stHMI_EL1008EcSlaveStateBits.bAdditionalLink
        Rectangle (2,364 85x18), "Port A", colour toggle: g_stHMI_EL1008EcSlaveStateBits.bPortA
        Rectangle (2,384 85x18), "Port B", colour toggle: g_stHMI_EL1008EcSlaveStateBits.bPortB
        Rectangle (2,404 85x18), "Port C", colour toggle: g_stHMI_EL1008EcSlaveStateBits.bPortC
        Rectangle (2,424 85x18), "Port D", colour toggle: g_stHMI_EL1008EcSlaveStateBits.bPortD
    Group (447,42 89x451)
        RoundedRectangle (0,2 89x449)
        Label (2,0 85x25), "EL2008"
        Rectangle (2,19 85x22), "Sftw Rev: %s", text variable: g_iHMI_ProdCodeEL2008
        Rectangle (2,39 85x22), "Port A CRC: %s", text variable: g_stHMI_EL2008CrcErrorEx.portA
        Rectangle (2,59 85x22), "Port B CRC: %s", text variable: g_stHMI_EL2008CrcErrorEx.portB
        Rectangle (2,79 85x22), "Port C CRC: %s", text variable: g_stHMI_EL2008CrcErrorEx.portC
        Rectangle (2,99 85x22), "Port D CRC: %s", text variable: g_stHMI_EL2008CrcErrorEx.portD
        Rectangle (2,124 85x18), "BootStrap", colour toggle: g_stHMI_EL2008EcSlaveStateBits.bBootStrap
        Rectangle (2,144 85x18), "Init", colour toggle: g_stHMI_EL2008EcSlaveStateBits.bInit
        Rectangle (2,164 85x18), "PreOP", colour toggle: g_stHMI_EL2008EcSlaveStateBits.bPreop
        Rectangle (2,184 85x18), "SafeOP", colour toggle: g_stHMI_EL2008EcSlaveStateBits.bSafeOp
        Rectangle (2,204 85x18), "OP", colour toggle: g_stHMI_EL2008EcSlaveStateBits.bOp
        Rectangle (2,224 85x18), "Error", colour toggle: g_stHMI_EL2008EcSlaveStateBits.bError
        Rectangle (2,244 85x18), "InvVPRS", colour toggle: g_stHMI_EL2008EcSlaveStateBits.bInvVPRS
        Rectangle (2,264 85x18), "InitCmdError", colour toggle: g_stHMI_EL2008EcSlaveStateBits.bInitCmdError
        Rectangle (2,284 85x18), "LinkNotPresent", colour toggle: g_stHMI_EL2008EcSlaveStateBits.bLinkNotPresent
        Rectangle (2,304 85x18), "Link_w/o_Com", colour toggle: g_stHMI_EL2008EcSlaveStateBits.bLinkWithoutComm
        Rectangle (2,324 85x18), "LinkMissing", colour toggle: g_stHMI_EL2008EcSlaveStateBits.bLinkMissing
        Rectangle (2,344 85x18), "AdditionalLink", colour toggle: g_stHMI_EL2008EcSlaveStateBits.bAdditionalLink
        Rectangle (2,364 85x18), "Port A", colour toggle: g_stHMI_EL2008EcSlaveStateBits.bPortA
        Rectangle (2,384 85x18), "Port B", colour toggle: g_stHMI_EL2008EcSlaveStateBits.bPortB
        Rectangle (2,404 85x18), "Port C", colour toggle: g_stHMI_EL2008EcSlaveStateBits.bPortC
        Rectangle (2,424 85x18), "Port D", colour toggle: g_stHMI_EL2008EcSlaveStateBits.bPortD
    Group (536,42 89x451)
        RoundedRectangle (0,2 89x449)
        Label (2,0 85x25), "EL3002"
        Rectangle (2,19 85x22), "Sftw Rev: %s", text variable: g_iHMI_ProdCodeEL3002
        Rectangle (2,39 85x22), "Port A CRC: %s", text variable: g_stHMI_EL3002CrcErrorEx.portA
        Rectangle (2,59 85x22), "Port B CRC: %s", text variable: g_stHMI_EL3002CrcErrorEx.portB
        Rectangle (2,79 85x22), "Port C CRC: %s", text variable: g_stHMI_EL3002CrcErrorEx.portC
        Rectangle (2,99 85x22), "Port D CRC: %s", text variable: g_stHMI_EL3002CrcErrorEx.portD
        Rectangle (2,124 85x18), "BootStrap", colour toggle: g_stHMI_EL3002EcSlaveStateBits.bBootStrap
        Rectangle (2,144 85x18), "Init", colour toggle: g_stHMI_EL3002EcSlaveStateBits.bInit
        Rectangle (2,164 85x18), "PreOP", colour toggle: g_stHMI_EL3002EcSlaveStateBits.bPreop
        Rectangle (2,184 85x18), "SafeOP", colour toggle: g_stHMI_EL3002EcSlaveStateBits.bSafeOp
        Rectangle (2,204 85x18), "OP", colour toggle: g_stHMI_EL3002EcSlaveStateBits.bOp
        Rectangle (2,224 85x18), "Error", colour toggle: g_stHMI_EL3002EcSlaveStateBits.bError
        Rectangle (2,244 85x18), "InvVPRS", colour toggle: g_stHMI_EL3002EcSlaveStateBits.bInvVPRS
        Rectangle (2,264 85x18), "InitCmdError", colour toggle: g_stHMI_EL3002EcSlaveStateBits.bInitCmdError
        Rectangle (2,284 85x18), "LinkNotPresent", colour toggle: g_stHMI_EL3002EcSlaveStateBits.bLinkNotPresent
        Rectangle (2,304 85x18), "Link_w/o_Com", colour toggle: g_stHMI_EL3002EcSlaveStateBits.bLinkWithoutComm
        Rectangle (2,324 85x18), "LinkMissing", colour toggle: g_stHMI_EL3002EcSlaveStateBits.bLinkMissing
        Rectangle (2,344 85x18), "AdditionalLink", colour toggle: g_stHMI_EL3002EcSlaveStateBits.bAdditionalLink
        Rectangle (2,364 85x18), "Port A", colour toggle: g_stHMI_EL3002EcSlaveStateBits.bPortA
        Rectangle (2,384 85x18), "Port B", colour toggle: g_stHMI_EL3002EcSlaveStateBits.bPortB
        Rectangle (2,404 85x18), "Port C", colour toggle: g_stHMI_EL3002EcSlaveStateBits.bPortC
        Rectangle (2,424 85x18), "Port D", colour toggle: g_stHMI_EL3002EcSlaveStateBits.bPortD
    RoundedRectangle (625,44 89x449)
    Label (627,42 85x25), "EL4032"
    Rectangle (627,61 85x22), "Sftw Rev: %s", text variable: g_iHMI_ProdCodeEL4032
    Rectangle (627,81 85x22), "Port A CRC: %s", text variable: g_stHMI_EL4032CrcErrorEx.portA
    Rectangle (627,101 85x22), "Port B CRC: %s", text variable: g_stHMI_EL4032CrcErrorEx.portB
    Rectangle (628,121 85x22), "Port C CRC: %s", text variable: g_stHMI_EL4032CrcErrorEx.portC
    Rectangle (628,141 85x22), "Port D CRC: %s", text variable: g_stHMI_EL4032CrcErrorEx.portD
    Rectangle (627,166 85x18), "BootStrap", colour toggle: g_stHMI_EL4032EcSlaveStateBits.bBootStrap
    Rectangle (627,186 85x18), "Init", colour toggle: g_stHMI_EL4032EcSlaveStateBits.bInit
    Rectangle (627,206 85x18), "PreOP", colour toggle: g_stHMI_EL4032EcSlaveStateBits.bPreop
    Rectangle (627,226 85x18), "SafeOP", colour toggle: g_stHMI_EL4032EcSlaveStateBits.bSafeOp
    Rectangle (627,246 85x18), "OP", colour toggle: g_stHMI_EL4032EcSlaveStateBits.bOp
    Rectangle (627,266 85x18), "Error", colour toggle: g_stHMI_EL4032EcSlaveStateBits.bError
    Rectangle (627,286 85x18), "InvVPRS", colour toggle: g_stHMI_EL4032EcSlaveStateBits.bInvVPRS
    Rectangle (627,306 85x18), "InitCmdError", colour toggle: g_stHMI_EL4032EcSlaveStateBits.bInitCmdError
    Rectangle (627,326 85x18), "LinkNotPresent", colour toggle: g_stHMI_EL4032EcSlaveStateBits.bLinkNotPresent
    Rectangle (627,346 85x18), "Link_w/o_Com", colour toggle: g_stHMI_EL4032EcSlaveStateBits.bLinkWithoutComm
    Rectangle (627,366 85x18), "LinkMissing", colour toggle: g_stHMI_EL4032EcSlaveStateBits.bLinkMissing
    Rectangle (627,386 85x18), "AdditionalLink", colour toggle: g_stHMI_EL4032EcSlaveStateBits.bAdditionalLink
    Rectangle (627,406 85x18), "Port A", colour toggle: g_stHMI_EL4032EcSlaveStateBits.bPortA
    Rectangle (627,426 85x18), "Port B", colour toggle: g_stHMI_EL4032EcSlaveStateBits.bPortB
    Rectangle (627,446 85x18), "Port C", colour toggle: g_stHMI_EL4032EcSlaveStateBits.bPortC
    Rectangle (627,466 85x18), "Port D", colour toggle: g_stHMI_EL4032EcSlaveStateBits.bPortD
    Group (714,42 89x451)
        RoundedRectangle (0,2 89x449)
        Label (2,0 85x25), "EL7201 #1"
        Rectangle (2,19 85x22), "Sftw Rev: %s", text variable: g_iHMI_ProdCodeEL7201_1
        Rectangle (2,39 85x22), "Port A CRC: %s", text variable: g_stHMI_EL7201_1CrcErrorEx.portA
        Rectangle (2,59 85x22), "Port B CRC: %s", text variable: g_stHMI_EL7201_1CrcErrorEx.portB
        Rectangle (2,79 85x22), "Port C CRC: %s", text variable: g_stHMI_EL7201_1CrcErrorEx.portC
        Rectangle (2,99 85x22), "Port D CRC: %s", text variable: g_stHMI_EL7201_1CrcErrorEx.portD
        Rectangle (2,124 85x18), "BootStrap", colour toggle: g_stHMI_EL7201_1EcSlaveStateBits.bBootStrap
        Rectangle (2,144 85x18), "Init", colour toggle: g_stHMI_EL7201_1EcSlaveStateBits.bInit
        Rectangle (2,164 85x18), "PreOP", colour toggle: g_stHMI_EL7201_1EcSlaveStateBits.bPreop
        Rectangle (2,184 85x18), "SafeOP", colour toggle: g_stHMI_EL7201_1EcSlaveStateBits.bSafeOp
        Rectangle (2,204 85x18), "OP", colour toggle: g_stHMI_EL7201_1EcSlaveStateBits.bOp
        Rectangle (2,224 85x18), "Error", colour toggle: g_stHMI_EL7201_1EcSlaveStateBits.bError
        Rectangle (2,244 85x18), "InvVPRS", colour toggle: g_stHMI_EL7201_1EcSlaveStateBits.bInvVPRS
        Rectangle (2,264 85x18), "InitCmdError", colour toggle: g_stHMI_EL7201_1EcSlaveStateBits.bInitCmdError
        Rectangle (2,284 85x18), "LinkNotPresent", colour toggle: g_stHMI_EL7201_1EcSlaveStateBits.bLinkNotPresent
        Rectangle (2,304 85x18), "Link_w/o_Com", colour toggle: g_stHMI_EL7201_1EcSlaveStateBits.bLinkWithoutComm
        Rectangle (2,324 85x18), "LinkMissing", colour toggle: g_stHMI_EL7201_1EcSlaveStateBits.bLinkMissing
        Rectangle (2,344 85x18), "AdditionalLink", colour toggle: g_stHMI_EL7201_1EcSlaveStateBits.bAdditionalLink
        Rectangle (2,364 85x18), "Port A", colour toggle: g_stHMI_EL7201_1EcSlaveStateBits.bPortA
        Rectangle (2,384 85x18), "Port B", colour toggle: g_stHMI_EL7201_1EcSlaveStateBits.bPortB
        Rectangle (2,404 85x18), "Port C", colour toggle: g_stHMI_EL7201_1EcSlaveStateBits.bPortC
        Rectangle (2,424 85x18), "Port D", colour toggle: g_stHMI_EL7201_1EcSlaveStateBits.bPortD
    Group (803,42 89x451)
        RoundedRectangle (0,2 89x449)
        Label (2,0 85x25), "EL7201 #2"
        Rectangle (2,19 85x22), "Sftw Rev: %s", text variable: g_iHMI_ProdCodeEL7201_2
        Rectangle (2,39 85x22), "Port A CRC: %s", text variable: g_stHMI_EL7201_2CrcErrorEx.portA
        Rectangle (2,59 85x22), "Port B CRC: %s", text variable: g_stHMI_EL7201_2CrcErrorEx.portB
        Rectangle (2,79 85x22), "Port C CRC: %s", text variable: g_stHMI_EL7201_2CrcErrorEx.portC
        Rectangle (2,99 85x22), "Port D CRC: %s", text variable: g_stHMI_EL7201_2CrcErrorEx.portD
        Rectangle (2,124 85x18), "BootStrap", colour toggle: g_stHMI_EL7201_2EcSlaveStateBits.bBootStrap
        Rectangle (2,144 85x18), "Init", colour toggle: g_stHMI_EL7201_2EcSlaveStateBits.bInit
        Rectangle (2,164 85x18), "PreOP", colour toggle: g_stHMI_EL7201_2EcSlaveStateBits.bPreop
        Rectangle (2,184 85x18), "SafeOP", colour toggle: g_stHMI_EL7201_2EcSlaveStateBits.bSafeOp
        Rectangle (2,204 85x18), "OP", colour toggle: g_stHMI_EL7201_2EcSlaveStateBits.bOp
        Rectangle (2,224 85x18), "Error", colour toggle: g_stHMI_EL7201_2EcSlaveStateBits.bError
        Rectangle (2,244 85x18), "InvVPRS", colour toggle: g_stHMI_EL7201_2EcSlaveStateBits.bInvVPRS
        Rectangle (2,264 85x18), "InitCmdError", colour toggle: g_stHMI_EL7201_2EcSlaveStateBits.bInitCmdError
        Rectangle (2,284 85x18), "LinkNotPresent", colour toggle: g_stHMI_EL7201_2EcSlaveStateBits.bLinkNotPresent
        Rectangle (2,304 85x18), "Link_w/o_Com", colour toggle: g_stHMI_EL7201_2EcSlaveStateBits.bLinkWithoutComm
        Rectangle (2,324 85x18), "LinkMissing", colour toggle: g_stHMI_EL7201_2EcSlaveStateBits.bLinkMissing
        Rectangle (2,344 85x18), "AdditionalLink", colour toggle: g_stHMI_EL7201_2EcSlaveStateBits.bAdditionalLink
        Rectangle (2,364 85x18), "Port A", colour toggle: g_stHMI_EL7201_2EcSlaveStateBits.bPortA
        Rectangle (2,384 85x18), "Port B", colour toggle: g_stHMI_EL7201_2EcSlaveStateBits.bPortB
        Rectangle (2,404 85x18), "Port C", colour toggle: g_stHMI_EL7201_2EcSlaveStateBits.bPortC
        Rectangle (2,424 85x18), "Port D", colour toggle: g_stHMI_EL7201_2EcSlaveStateBits.bPortD
    Group (892,42 89x451)
        RoundedRectangle (0,2 89x449)
        Label (2,0 85x25), "EK1122"
        Rectangle (2,19 85x22), "Sftw Rev: %s", text variable: g_iHMI_ProdCodeEK1122
        Rectangle (2,39 85x22), "Port A CRC: %s", text variable: g_stHMI_EK1122_CrcErrorEx.portA
        Rectangle (2,59 85x22), "Port B CRC: %s", text variable: g_stHMI_EK1122_CrcErrorEx.portB
        Rectangle (2,79 85x22), "Port C CRC: %s", text variable: g_stHMI_EK1122_CrcErrorEx.portC
        Rectangle (2,99 85x22), "Port D CRC: %s", text variable: g_stHMI_EK1122_CrcErrorEx.portD
        Rectangle (2,124 85x18), "BootStrap", colour toggle: g_stHMI_EK1122_EcSlaveStateBits.bBootStrap
        Rectangle (2,144 85x18), "Init", colour toggle: g_stHMI_EK1122_EcSlaveStateBits.bInit
        Rectangle (2,164 85x18), "PreOP", colour toggle: g_stHMI_EK1122_EcSlaveStateBits.bPreop
        Rectangle (2,184 85x18), "SafeOP", colour toggle: g_stHMI_EK1122_EcSlaveStateBits.bSafeOp
        Rectangle (2,204 85x18), "OP", colour toggle: g_stHMI_EK1122_EcSlaveStateBits.bOp
        Rectangle (2,224 85x18), "Error", colour toggle: g_stHMI_EK1122_EcSlaveStateBits.bError
        Rectangle (2,244 85x18), "InvVPRS", colour toggle: g_stHMI_EK1122_EcSlaveStateBits.bInvVPRS
        Rectangle (2,264 85x18), "InitCmdError", colour toggle: g_stHMI_EK1122_EcSlaveStateBits.bInitCmdError
        Rectangle (2,284 85x18), "LinkNotPresent", colour toggle: g_stHMI_EK1122_EcSlaveStateBits.bLinkNotPresent
        Rectangle (2,304 85x18), "Link_w/o_Com", colour toggle: g_stHMI_EK1122_EcSlaveStateBits.bLinkWithoutComm
        Rectangle (2,324 85x18), "LinkMissing", colour toggle: g_stHMI_EK1122_EcSlaveStateBits.bLinkMissing
        Rectangle (2,344 85x18), "AdditionalLink", colour toggle: g_stHMI_EK1122_EcSlaveStateBits.bAdditionalLink
        Rectangle (2,364 85x18), "Port A", colour toggle: g_stHMI_EK1122_EcSlaveStateBits.bPortA
        Rectangle (2,384 85x18), "Port B", colour toggle: g_stHMI_EK1122_EcSlaveStateBits.bPortB
        Rectangle (2,404 85x18), "Port C", colour toggle: g_stHMI_EK1122_EcSlaveStateBits.bPortC
        Rectangle (2,424 85x18), "Port D", colour toggle: g_stHMI_EK1122_EcSlaveStateBits.bPortD
END_VISUALIZATION

// ---- VISUs/MDP_MainboardCPUMemory.TcVIS
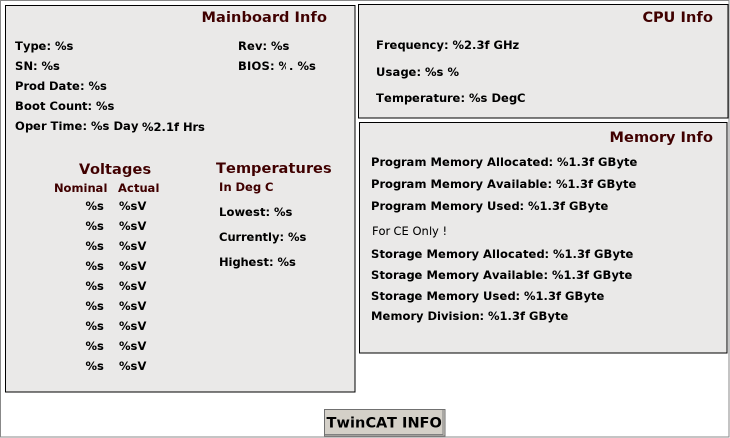
VISUALIZATION MDP_MainboardCPUMemory  // 730x438
    RoundedRectangle (358,4 370x114)
    RoundedRectangle (5,5 350x387)
    Label (192,4 145x26), "Mainboard Info"
    Rectangle (12,35 141x22), "Type: %s", text variable: g_sHMI_MainboardType
    Rectangle (12,55 171x22), "SN: %s", text variable: g_sHMI_MainboardSN
    Rectangle (12,75 207x22), "Prod Date: %s", text variable: g_sHMI_MainboardProdDate
    Rectangle (12,95 151x22), "Boot Count: %s", text variable: g_udiHMI_MainboardBootCount
    Rectangle (12,115 184x22), "Oper Time: %s Days", text variable: g_udiHMI_MainboardOperTimeDays
    Rectangle (139,116 70x22), "%2.1f Hrs", text variable: g_lrHMI_MainboardOperTimeHrs
    Label (213,155 120x26), "Temperatures"
    Rectangle (216,201 102x22), "Lowest: %s", text variable: g_diHMI_MainboardMinTemp
    Rectangle (216,226 102x22), "Currently: %s", text variable: g_iHMI_MainboardActualTemp
    Rectangle (216,251 102x22), "Highest: %s", text variable: g_diHMI_MainboardMaxTemp
    Rectangle (235,35 67x22), "Rev: %s", text variable: g_bHMI_MainboardRevision
    Rectangle (235,55 67x22), "BIOS: %s", text variable: g_bHMI_MainboardBiosMajVers
    Rectangle (286,55 67x22), ". %s", text variable: g_bHMI_MainboardBiosMinVers
    Label (51,175 76x26), "Nominal"
    Rectangle (37,195 70x22), "%s", text variable: g_sHMI_Mainboard1p05v
    Rectangle (37,215 70x22), "%s", text variable: g_sHMI_MainboardVccCore
    Rectangle (37,235 70x22), "%s", text variable: g_sHMI_Mainboard5v
    Rectangle (37,255 70x22), "%s", text variable: g_sHMI_Mainboard12v
    Rectangle (37,275 70x22), "%s", text variable: g_sHMI_MainboardVBatt
    Rectangle (16,295 91x22), "%s", text variable: g_sHMI_MainboardPwrCtrlVcc
    Rectangle (16,315 91x22), "%s", text variable: g_sHMI_MainboardCX2100_5v
    Rectangle (18,335 89x22), "%s", text variable: g_sHMI_MainboardCX2100_12v
    Rectangle (19,355 88x22), "%s", text variable: g_sHMI_MainboardCX2100_24v
    Label (115,175 76x26), "Actual"
    Rectangle (116,195 70x22), "%sV", text variable: g_lrHMI_Mainboard1p05v
    Rectangle (116,215 70x22), "%sV", text variable: g_lrHMI_MainboardVccCore
    Rectangle (116,235 70x22), "%sV", text variable: g_lrHMI_Mainboard5v
    Rectangle (116,255 70x22), "%sV", text variable: g_lrHMI_Mainboard12v
    Rectangle (116,275 70x22), "%sV", text variable: g_lrHMI_MainboardVBatt
    Rectangle (116,295 91x22), "%sV", text variable: g_lrHMI_MainboardPwrCtrlVcc
    Rectangle (116,315 91x22), "%sV", text variable: g_lrHMI_MainboardCX2100_5v
    Rectangle (116,335 89x22), "%sV", text variable: g_lrHMI_MainboardCX2100_12v
    Rectangle (116,355 88x22), "%sV", text variable: g_lrHMI_MainboardCX2100_24v
    Label (76,156 81x26), "Voltages"
    Label (216,174 120x26), "In Deg C"
    Label (596,4 120x26), "CPU Info"
    Rectangle (373,34 163x22), "Frequency: %2.3f GHz", text variable: g_lrHMI_CPUfrequency
    Rectangle (373,61 122x22), "Usage: %s %", text variable: g_iHMI_CPUusage
    Rectangle (373,87 156x22), "Temperature: %s DegC", text variable: g_iHMI_CPUtemperature
    Button (324,409 121x27), "TwinCAT INFO"
        OnMouseClick: change screen: TwinCAT_INFO
    RoundedRectangle (359,122 368x231)
    Label (596,124 120x26), "Memory Info"
    Rectangle (368,151 289x22), "Program Memory Allocated: %1.3f GByte", text variable: g_lrHMI_ProgMemAllocated_InGB
    Rectangle (368,173 287x22), "Program Memory Available: %1.3f GByte", text variable: g_lrHMI_ProgMemAvailable_InGB
    Rectangle (368,243 289x22), "Storage Memory Allocated: %1.3f GByte", text variable: g_lrHMI_ProgStorAllocated_InGB
    Rectangle (368,264 289x22), "Storage Memory Available: %1.3f GByte", text variable: g_lrHMI_ProgStorAvailable_InGB
    Rectangle (368,305 289x22), "Memory Division: %1.3f GByte", text variable: g_lrHMI_ProgStorMemDivision_InGB
    Label (369,216 150x30), "For CE Only !"
    Rectangle (368,195 287x22), "Program Memory Used: %1.3f GByte", text variable: g_lrHMI_ProgMemUsed_InGB
    Rectangle (368,285 289x22), "Storage Memory Used: %1.3f GByte", text variable: g_lrHMI_ProgStorUsed_InGB
END_VISUALIZATION

// ---- VISUs/MDP_NicTime.TcVIS
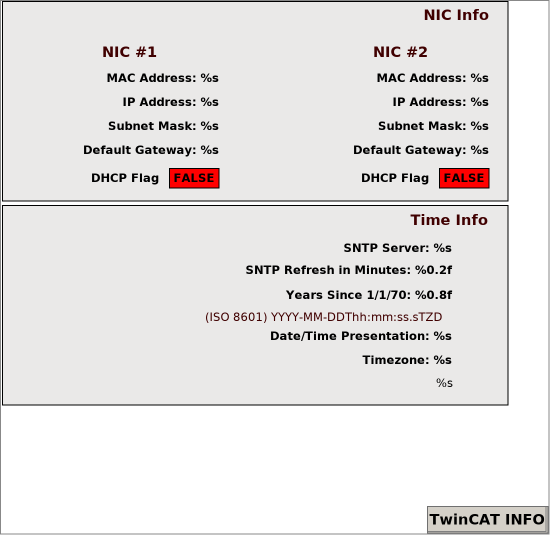
VISUALIZATION MDP_NicTime  // 550x535
    RoundedRectangle (2,1 506x200)
    Rectangle (7,67 215x22), "MAC Address: %s", text variable: System_Functions.ST_NIC0_ModContent.sMACAddress
    Rectangle (9,91 213x22), "IP Address: %s", text variable: System_Functions.ST_NIC0_ModContent.sIPAddress
    Rectangle (11,115 211x22), "Subnet Mask: %s", text variable: System_Functions.ST_NIC0_ModContent.sSubnetMask
    Rectangle (14,139 208x22), "Default Gateway: %s", text variable: System_Functions.ST_NIC0_ModContent.sDefaultGateway
    Group (169,168 50x20)
        Rectangle (0,0 50x20), "TRUE", invisible if: NOT System_Functions.ST_NIC0_ModContent.xDHCP
        Rectangle (0,0 50x20), "FALSE", invisible if: System_Functions.ST_NIC0_ModContent.xDHCP
    Label (77,166 85x24), "DHCP Flag"
    Rectangle (277,67 215x22), "MAC Address: %s", text variable: System_Functions.ST_NIC1_ModContent.sMACAddress
    Rectangle (279,91 213x22), "IP Address: %s", text variable: System_Functions.ST_NIC1_ModContent.sIPAddress
    Rectangle (281,115 211x22), "Subnet Mask: %s", text variable: System_Functions.ST_NIC1_ModContent.sSubnetMask
    Rectangle (284,139 208x22), "Default Gateway: %s", text variable: System_Functions.ST_NIC1_ModContent.sDefaultGateway
    Group (439,168 50x20)
        Rectangle (0,0 50x20), "TRUE", invisible if: NOT System_Functions.ST_NIC1_ModContent.xDHCP
        Rectangle (0,0 50x20), "FALSE", invisible if: System_Functions.ST_NIC1_ModContent.xDHCP
    Label (350,166 82x24), "DHCP Flag"
    Button (427,506 121x27), "TwinCAT INFO"
        OnMouseClick: change screen: TwinCAT_INFO
    Label (372,2 120x26), "NIC Info"
    Label (99,39 120x26), "NIC #1"
    Label (370,39 120x26), "NIC #2"
    RoundedRectangle (2,205 506x200)
    Label (371,207 120x26), "Time Info"
    Rectangle (10,237 445x22), "SNTP Server: %s", text variable: g_sHMI_SNTP_Server
    Rectangle (8,259 447x22), "SNTP Refresh in Minutes: %0.2f", text variable: g_lrHMI_SNTP_Refresh_Minutes
    Rectangle (10,284 445x22), "Years Since 1/1/70: %0.8f", text variable: g_lrHMI_Years_Since_1_1_1970
    Rectangle (9,325 446x22), "Date/Time Presentation: %s", text variable: System_Functions.ST_NIC0_ModContent.sMACAddress
    Rectangle (6,349 449x22), "Timezone: %s", text variable: System_Functions.ST_NIC0_ModContent.sMACAddress
    Label (202,304 274x26), "(ISO 8601) YYYY-MM-DDThh:mm:ss.sTZD"
    Rectangle (15,368 441x30), "%s", text variable: g_sHMI_CurrentTimeZone
END_VISUALIZATION

// ---- VISUs/TwinCAT_INFO.TcVIS
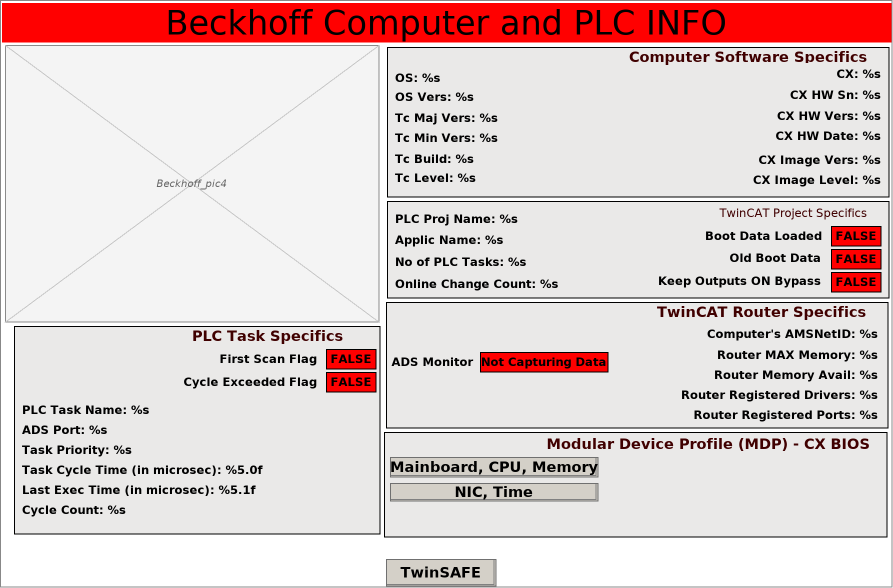
VISUALIZATION TwinCAT_INFO  // 893x588
    RoundedRectangle (384,432 503x105)
    Button (386,559 110x27), "TwinSAFE"
        OnMouseClick: change screen: TwinSAFE
    RoundedRectangle (2,3 889x39), "Beckhoff Computer and PLC INFO"
    RoundedRectangle (387,47 502x150)
    Label (614,44 256x26), "Computer Software Specifics"
    Rectangle (392,67 256x22), "OS: %s", text variable: g_stHMI_DevIdent.strImageOsName
    RoundedRectangle (387,201 502x97)
    Label (695,200 175x26), "TwinCAT Project Specifics"
    RoundedRectangle (386,302 502x126)
    Label (613,299 256x26), "TwinCAT Router Specifics"
    RoundedRectangle (14,326 366x208)
    Label (188,323 158x26), "PLC Task Specifics"
    Rectangle (392,86 208x22), "OS Vers: %s", text variable: g_stHMI_DevIdent.strImageOsVersion
    Rectangle (392,107 119x22), "Tc Maj Vers: %s", text variable: g_stHMI_DevIdent.strTwinCATVersion
    Rectangle (392,127 111x22), "Tc Min Vers: %s", text variable: g_stHMI_DevIdent.strTwinCATRevision
    Rectangle (392,148 111x22), "Tc Build: %s", text variable: g_stHMI_DevIdent.strTwinCATBuild
    Rectangle (392,167 111x22), "Tc Level: %s", text variable: g_stHMI_DevIdent.strTwinCATLevel
    Rectangle (738,63 146x22), "CX: %s", text variable: g_stHMI_DevIdent.strHardwareModel
    Rectangle (726,84 158x22), "CX HW Sn: %s", text variable: g_stHMI_DevIdent.strHardwareSerialNo
    Rectangle (733,105 151x22), "CX HW Vers: %s", text variable: g_stHMI_DevIdent.strHardwareVersion
    Rectangle (737,125 147x22), "CX HW Date: %s", text variable: g_stHMI_DevIdent.strHardwareDate
    Rectangle (725,149 159x22), "CX Image Vers: %s", text variable: g_stHMI_DevIdent.strImageVersion
    Rectangle (625,169 259x22), "CX Image Level: %s", text variable: g_stHMI_DevIdent.strImageLevel
    Rectangle (392,208 283x22), "PLC Proj Name: %s", text variable: g_stHMI_AppInfo.ProjectName
    Rectangle (392,229 359x22), "Applic Name: %s", text variable: g_stHMI_AppInfo.AppName
    Rectangle (392,251 155x22), "No of PLC Tasks: %s", text variable: g_stHMI_AppInfo.TaskCnt
    Rectangle (392,273 191x22), "Online Change Count: %s", text variable: g_stHMI_AppInfo.OnlineChangeCnt
    Group (831,226 50x20)
        Rectangle (0,0 50x20), "TRUE", invisible if: NOT g_stHMI_AppInfo.BootDataLoaded
        Rectangle (0,0 50x20), "FALSE", invisible if: g_stHMI_AppInfo.BootDataLoaded
    Label (705,224 120x24), "Boot Data Loaded"
    Group (831,249 50x20)
        Rectangle (0,0 50x20), "TRUE", invisible if: NOT g_stHMI_AppInfo.OldBootData
        Rectangle (0,0 50x20), "FALSE", invisible if: g_stHMI_AppInfo.OldBootData
    Label (726,246 98x24), "Old Boot Data"
    Group (831,272 50x20)
        Rectangle (0,0 49x19), "TRUE", invisible if: NOT g_stHMI_AppInfo.KeepOutputsOnBP
        Rectangle (0,0 50x20), "FALSE", invisible if: g_stHMI_AppInfo.KeepOutputsOnBP
    Label (645,269 179x24), "Keep Outputs ON Bypass"
    Label (389,350 87x24), "ADS Monitor"
    Group (480,352 128x20)
        Rectangle (0,0 128x20), "Capturing Data", invisible if: NOT g_stHMI_RouterStatusInfo.amsDebugLog
        Rectangle (0,0 128x20), "Not Capturing Data", invisible if: g_stHMI_RouterStatusInfo.amsDebugLog
    Rectangle (560,323 321x22), "Computer's AMSNetID: %s", text variable: g_stHMI_DevIdent.strAmsNetId
    Rectangle (673,344 208x22), "Router MAX Memory: %s", text variable: g_stHMI_RouterStatusInfo.maxMem
    Rectangle (673,364 208x22), "Router Memory Avail: %s", text variable: g_stHMI_RouterStatusInfo.maxMemAvail
    Rectangle (673,384 208x22), "Router Registered Drivers: %s", text variable: g_stHMI_RouterStatusInfo.regDrivers
    Rectangle (673,404 208x22), "Router Registered Ports: %s", text variable: g_stHMI_RouterStatusInfo.regPorts
    Group (326,349 50x20)
        Rectangle (0,0 50x20), "TRUE", invisible if: NOT g_stHMI_PlcTaskSystemInfo.FirstCycle
        Rectangle (0,0 50x20), "FALSE", invisible if: g_stHMI_PlcTaskSystemInfo.FirstCycle
    Label (200,347 120x24), "First Scan Flag"
    Group (326,372 50x20)
        Rectangle (0,0 50x20), "TRUE", invisible if: NOT g_stHMI_PlcTaskSystemInfo.CycleTimeExceeded
        Rectangle (0,0 50x20), "FALSE", invisible if: g_stHMI_PlcTaskSystemInfo.CycleTimeExceeded
    Label (178,370 142x24), "Cycle Exceeded Flag"
    Rectangle (19,399 357x22), "PLC Task Name: %s", text variable: g_stHMI_PlcTaskSystemInfo.TaskName
    Rectangle (19,419 299x22), "ADS Port: %s", text variable: g_stHMI_PlcTaskSystemInfo.AdsPort
    Rectangle (19,439 214x22), "Task Priority: %s", text variable: g_stHMI_PlcTaskSystemInfo.Priority
    Rectangle (19,459 298x22), "Task Cycle Time (in microsec): %5.0f", text variable: g_lrHMI_PlcTaskSystemInfo_CycleTime
    Rectangle (19,479 298x22), "Last Exec Time (in microsec): %5.1f", text variable: g_lrHMI_PlcTaskSystemInfo_LastExecTime
    Rectangle (19,499 214x22), "Cycle Count: %s", text variable: g_stHMI_PlcTaskSystemInfo.CycleCount
    Button (390,483 208x18), "NIC, Time"
        OnMouseClick: change screen: MDP_NicTime
    Button (390,457 208x20), "Mainboard, CPU, Memory"
        OnMouseClick: change screen: MDP_MainboardCPUMemory
    Label (516,431 357x26), "Modular Device Profile (MDP) - CX BIOS"
    Image (5,45 374x277), image: Beckhoff_pic4
END_VISUALIZATION

// ---- VISUs/TwinCAT_INFO.TcVIS
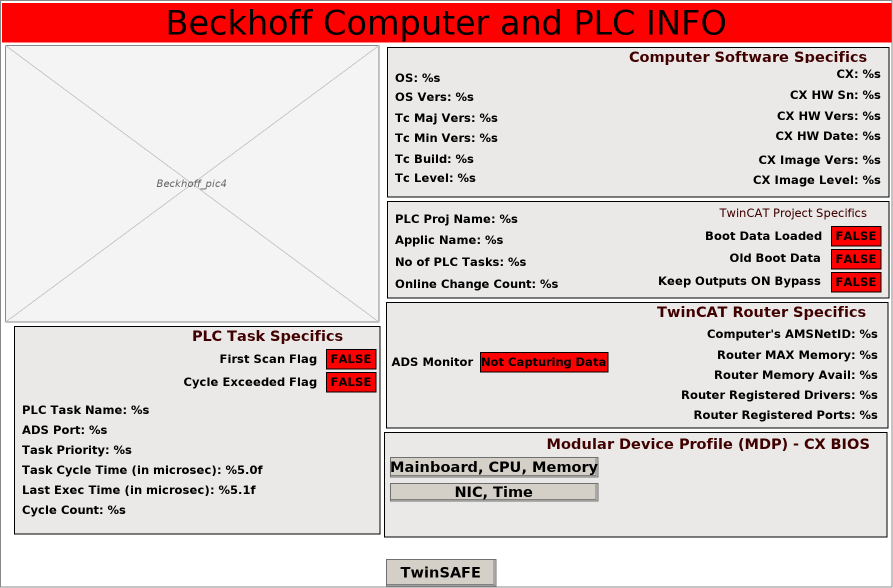
VISUALIZATION TwinCAT_INFO  // 893x588
    RoundedRectangle (384,432 503x105)
    Button (386,559 110x27), "TwinSAFE"
        OnMouseClick: change screen: TwinSAFE
    RoundedRectangle (2,3 889x39), "Beckhoff Computer and PLC INFO"
    RoundedRectangle (387,47 502x150)
    Label (614,44 256x26), "Computer Software Specifics"
    Rectangle (392,67 256x22), "OS: %s", text variable: g_stHMI_DevIdent.strImageOsName
    RoundedRectangle (387,201 502x97)
    Label (695,200 175x26), "TwinCAT Project Specifics"
    RoundedRectangle (386,302 502x126)
    Label (613,299 256x26), "TwinCAT Router Specifics"
    RoundedRectangle (14,326 366x208)
    Label (188,323 158x26), "PLC Task Specifics"
    Rectangle (392,86 208x22), "OS Vers: %s", text variable: g_stHMI_DevIdent.strImageOsVersion
    Rectangle (392,107 119x22), "Tc Maj Vers: %s", text variable: g_stHMI_DevIdent.strTwinCATVersion
    Rectangle (392,127 111x22), "Tc Min Vers: %s", text variable: g_stHMI_DevIdent.strTwinCATRevision
    Rectangle (392,148 111x22), "Tc Build: %s", text variable: g_stHMI_DevIdent.strTwinCATBuild
    Rectangle (392,167 111x22), "Tc Level: %s", text variable: g_stHMI_DevIdent.strTwinCATLevel
    Rectangle (738,63 146x22), "CX: %s", text variable: g_stHMI_DevIdent.strHardwareModel
    Rectangle (726,84 158x22), "CX HW Sn: %s", text variable: g_stHMI_DevIdent.strHardwareSerialNo
    Rectangle (733,105 151x22), "CX HW Vers: %s", text variable: g_stHMI_DevIdent.strHardwareVersion
    Rectangle (737,125 147x22), "CX HW Date: %s", text variable: g_stHMI_DevIdent.strHardwareDate
    Rectangle (725,149 159x22), "CX Image Vers: %s", text variable: g_stHMI_DevIdent.strImageVersion
    Rectangle (625,169 259x22), "CX Image Level: %s", text variable: g_stHMI_DevIdent.strImageLevel
    Rectangle (392,208 283x22), "PLC Proj Name: %s", text variable: g_stHMI_AppInfo.ProjectName
    Rectangle (392,229 359x22), "Applic Name: %s", text variable: g_stHMI_AppInfo.AppName
    Rectangle (392,251 155x22), "No of PLC Tasks: %s", text variable: g_stHMI_AppInfo.TaskCnt
    Rectangle (392,273 191x22), "Online Change Count: %s", text variable: g_stHMI_AppInfo.OnlineChangeCnt
    Group (831,226 50x20)
        Rectangle (0,0 50x20), "TRUE", invisible if: NOT g_stHMI_AppInfo.BootDataLoaded
        Rectangle (0,0 50x20), "FALSE", invisible if: g_stHMI_AppInfo.BootDataLoaded
    Label (705,224 120x24), "Boot Data Loaded"
    Group (831,249 50x20)
        Rectangle (0,0 50x20), "TRUE", invisible if: NOT g_stHMI_AppInfo.OldBootData
        Rectangle (0,0 50x20), "FALSE", invisible if: g_stHMI_AppInfo.OldBootData
    Label (726,246 98x24), "Old Boot Data"
    Group (831,272 50x20)
        Rectangle (0,0 49x19), "TRUE", invisible if: NOT g_stHMI_AppInfo.KeepOutputsOnBP
        Rectangle (0,0 50x20), "FALSE", invisible if: g_stHMI_AppInfo.KeepOutputsOnBP
    Label (645,269 179x24), "Keep Outputs ON Bypass"
    Label (389,350 87x24), "ADS Monitor"
    Group (480,352 128x20)
        Rectangle (0,0 128x20), "Capturing Data", invisible if: NOT g_stHMI_RouterStatusInfo.amsDebugLog
        Rectangle (0,0 128x20), "Not Capturing Data", invisible if: g_stHMI_RouterStatusInfo.amsDebugLog
    Rectangle (560,323 321x22), "Computer's AMSNetID: %s", text variable: g_stHMI_DevIdent.strAmsNetId
    Rectangle (673,344 208x22), "Router MAX Memory: %s", text variable: g_stHMI_RouterStatusInfo.maxMem
    Rectangle (673,364 208x22), "Router Memory Avail: %s", text variable: g_stHMI_RouterStatusInfo.maxMemAvail
    Rectangle (673,384 208x22), "Router Registered Drivers: %s", text variable: g_stHMI_RouterStatusInfo.regDrivers
    Rectangle (673,404 208x22), "Router Registered Ports: %s", text variable: g_stHMI_RouterStatusInfo.regPorts
    Group (326,349 50x20)
        Rectangle (0,0 50x20), "TRUE", invisible if: NOT g_stHMI_PlcTaskSystemInfo.FirstCycle
        Rectangle (0,0 50x20), "FALSE", invisible if: g_stHMI_PlcTaskSystemInfo.FirstCycle
    Label (200,347 120x24), "First Scan Flag"
    Group (326,372 50x20)
        Rectangle (0,0 50x20), "TRUE", invisible if: NOT g_stHMI_PlcTaskSystemInfo.CycleTimeExceeded
        Rectangle (0,0 50x20), "FALSE", invisible if: g_stHMI_PlcTaskSystemInfo.CycleTimeExceeded
    Label (178,370 142x24), "Cycle Exceeded Flag"
    Rectangle (19,399 357x22), "PLC Task Name: %s", text variable: g_stHMI_PlcTaskSystemInfo.TaskName
    Rectangle (19,419 299x22), "ADS Port: %s", text variable: g_stHMI_PlcTaskSystemInfo.AdsPort
    Rectangle (19,439 214x22), "Task Priority: %s", text variable: g_stHMI_PlcTaskSystemInfo.Priority
    Rectangle (19,459 298x22), "Task Cycle Time (in microsec): %5.0f", text variable: g_lrHMI_PlcTaskSystemInfo_CycleTime
    Rectangle (19,479 298x22), "Last Exec Time (in microsec): %5.1f", text variable: g_lrHMI_PlcTaskSystemInfo_LastExecTime
    Rectangle (19,499 214x22), "Cycle Count: %s", text variable: g_stHMI_PlcTaskSystemInfo.CycleCount
    Button (390,483 208x18), "NIC, Time"
        OnMouseClick: change screen: MDP_NicTime
    Button (390,457 208x20), "Mainboard, CPU, Memory"
        OnMouseClick: change screen: MDP_MainboardCPUMemory
    Label (516,431 357x26), "Modular Device Profile (MDP) - CX BIOS"
    Image (5,45 374x277), image: Beckhoff_pic4
END_VISUALIZATION

// ---- VISUs/TwinCAT_INFO.TcVIS
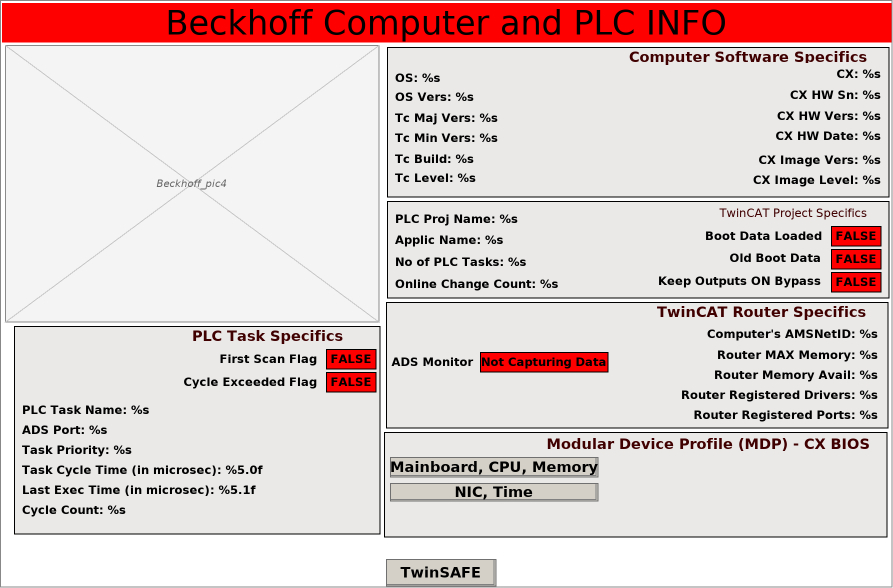
VISUALIZATION TwinCAT_INFO  // 893x588
    RoundedRectangle (384,432 503x105)
    Button (386,559 110x27), "TwinSAFE"
        OnMouseClick: change screen: TwinSAFE
    RoundedRectangle (2,3 889x39), "Beckhoff Computer and PLC INFO"
    RoundedRectangle (387,47 502x150)
    Label (614,44 256x26), "Computer Software Specifics"
    Rectangle (392,67 256x22), "OS: %s", text variable: g_stHMI_DevIdent.strImageOsName
    RoundedRectangle (387,201 502x97)
    Label (695,200 175x26), "TwinCAT Project Specifics"
    RoundedRectangle (386,302 502x126)
    Label (613,299 256x26), "TwinCAT Router Specifics"
    RoundedRectangle (14,326 366x208)
    Label (188,323 158x26), "PLC Task Specifics"
    Rectangle (392,86 208x22), "OS Vers: %s", text variable: g_stHMI_DevIdent.strImageOsVersion
    Rectangle (392,107 119x22), "Tc Maj Vers: %s", text variable: g_stHMI_DevIdent.strTwinCATVersion
    Rectangle (392,127 111x22), "Tc Min Vers: %s", text variable: g_stHMI_DevIdent.strTwinCATRevision
    Rectangle (392,148 111x22), "Tc Build: %s", text variable: g_stHMI_DevIdent.strTwinCATBuild
    Rectangle (392,167 111x22), "Tc Level: %s", text variable: g_stHMI_DevIdent.strTwinCATLevel
    Rectangle (738,63 146x22), "CX: %s", text variable: g_stHMI_DevIdent.strHardwareModel
    Rectangle (726,84 158x22), "CX HW Sn: %s", text variable: g_stHMI_DevIdent.strHardwareSerialNo
    Rectangle (733,105 151x22), "CX HW Vers: %s", text variable: g_stHMI_DevIdent.strHardwareVersion
    Rectangle (737,125 147x22), "CX HW Date: %s", text variable: g_stHMI_DevIdent.strHardwareDate
    Rectangle (725,149 159x22), "CX Image Vers: %s", text variable: g_stHMI_DevIdent.strImageVersion
    Rectangle (625,169 259x22), "CX Image Level: %s", text variable: g_stHMI_DevIdent.strImageLevel
    Rectangle (392,208 283x22), "PLC Proj Name: %s", text variable: g_stHMI_AppInfo.ProjectName
    Rectangle (392,229 359x22), "Applic Name: %s", text variable: g_stHMI_AppInfo.AppName
    Rectangle (392,251 155x22), "No of PLC Tasks: %s", text variable: g_stHMI_AppInfo.TaskCnt
    Rectangle (392,273 191x22), "Online Change Count: %s", text variable: g_stHMI_AppInfo.OnlineChangeCnt
    Group (831,226 50x20)
        Rectangle (0,0 50x20), "TRUE", invisible if: NOT g_stHMI_AppInfo.BootDataLoaded
        Rectangle (0,0 50x20), "FALSE", invisible if: g_stHMI_AppInfo.BootDataLoaded
    Label (705,224 120x24), "Boot Data Loaded"
    Group (831,249 50x20)
        Rectangle (0,0 50x20), "TRUE", invisible if: NOT g_stHMI_AppInfo.OldBootData
        Rectangle (0,0 50x20), "FALSE", invisible if: g_stHMI_AppInfo.OldBootData
    Label (726,246 98x24), "Old Boot Data"
    Group (831,272 50x20)
        Rectangle (0,0 49x19), "TRUE", invisible if: NOT g_stHMI_AppInfo.KeepOutputsOnBP
        Rectangle (0,0 50x20), "FALSE", invisible if: g_stHMI_AppInfo.KeepOutputsOnBP
    Label (645,269 179x24), "Keep Outputs ON Bypass"
    Label (389,350 87x24), "ADS Monitor"
    Group (480,352 128x20)
        Rectangle (0,0 128x20), "Capturing Data", invisible if: NOT g_stHMI_RouterStatusInfo.amsDebugLog
        Rectangle (0,0 128x20), "Not Capturing Data", invisible if: g_stHMI_RouterStatusInfo.amsDebugLog
    Rectangle (560,323 321x22), "Computer's AMSNetID: %s", text variable: g_stHMI_DevIdent.strAmsNetId
    Rectangle (673,344 208x22), "Router MAX Memory: %s", text variable: g_stHMI_RouterStatusInfo.maxMem
    Rectangle (673,364 208x22), "Router Memory Avail: %s", text variable: g_stHMI_RouterStatusInfo.maxMemAvail
    Rectangle (673,384 208x22), "Router Registered Drivers: %s", text variable: g_stHMI_RouterStatusInfo.regDrivers
    Rectangle (673,404 208x22), "Router Registered Ports: %s", text variable: g_stHMI_RouterStatusInfo.regPorts
    Group (326,349 50x20)
        Rectangle (0,0 50x20), "TRUE", invisible if: NOT g_stHMI_PlcTaskSystemInfo.FirstCycle
        Rectangle (0,0 50x20), "FALSE", invisible if: g_stHMI_PlcTaskSystemInfo.FirstCycle
    Label (200,347 120x24), "First Scan Flag"
    Group (326,372 50x20)
        Rectangle (0,0 50x20), "TRUE", invisible if: NOT g_stHMI_PlcTaskSystemInfo.CycleTimeExceeded
        Rectangle (0,0 50x20), "FALSE", invisible if: g_stHMI_PlcTaskSystemInfo.CycleTimeExceeded
    Label (178,370 142x24), "Cycle Exceeded Flag"
    Rectangle (19,399 357x22), "PLC Task Name: %s", text variable: g_stHMI_PlcTaskSystemInfo.TaskName
    Rectangle (19,419 299x22), "ADS Port: %s", text variable: g_stHMI_PlcTaskSystemInfo.AdsPort
    Rectangle (19,439 214x22), "Task Priority: %s", text variable: g_stHMI_PlcTaskSystemInfo.Priority
    Rectangle (19,459 298x22), "Task Cycle Time (in microsec): %5.0f", text variable: g_lrHMI_PlcTaskSystemInfo_CycleTime
    Rectangle (19,479 298x22), "Last Exec Time (in microsec): %5.1f", text variable: g_lrHMI_PlcTaskSystemInfo_LastExecTime
    Rectangle (19,499 214x22), "Cycle Count: %s", text variable: g_stHMI_PlcTaskSystemInfo.CycleCount
    Button (390,483 208x18), "NIC, Time"
        OnMouseClick: change screen: MDP_NicTime
    Button (390,457 208x20), "Mainboard, CPU, Memory"
        OnMouseClick: change screen: MDP_MainboardCPUMemory
    Label (516,431 357x26), "Modular Device Profile (MDP) - CX BIOS"
    Image (5,45 374x277), image: Beckhoff_pic4
END_VISUALIZATION

// ---- VISUs/TwinSAFE.TcVIS
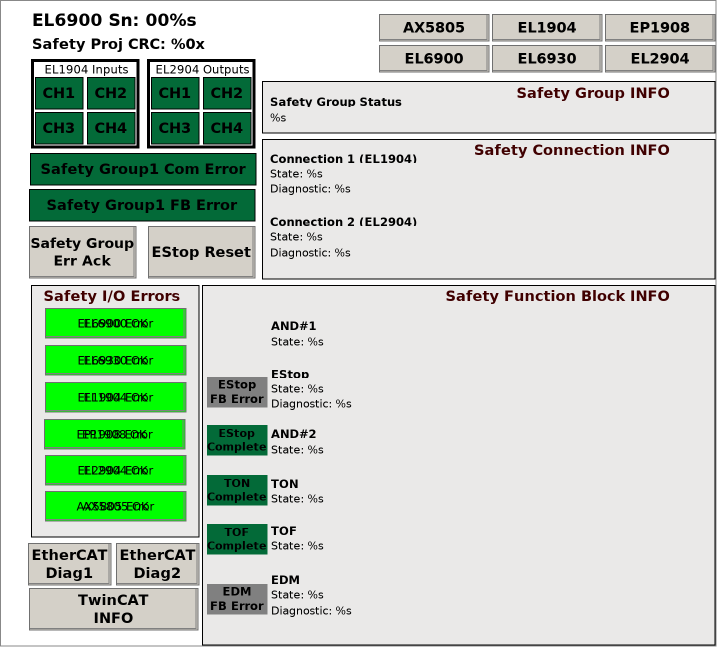
VISUALIZATION TwinSAFE  // 717x647
    RoundedRectangle (31,285 168x252)
    Rectangle (31,59 108x89)
    Rectangle (29,9 219x22), "EL6900 Sn: 00%s", text variable: g_udiHMI_SerialNumber
    Rectangle (29,33 232x22), "Safety Proj CRC: %0x", text variable: g_uiHMI_ProjectCRC
    Rectangle (35,77 48x32), "CH1", colour toggle: g_xHMI_EL1904Ch1
    Rectangle (87,77 48x32), "CH2", colour toggle: g_xHMI_EL1904Ch2
    Rectangle (35,112 48x32), "CH3", colour toggle: g_xHMI_EL1904Ch3
    Rectangle (87,112 48x32), "CH4", colour toggle: g_xHMI_EL1904Ch4
    Label (37,58 99x23), "EL1904 Inputs"
    Rectangle (147,59 108x89)
    Rectangle (151,77 48x32), "CH1", colour toggle: g_xHMI_EL2904Ch1
    Rectangle (203,77 48x32), "CH2", colour toggle: g_xHMI_EL2904Ch2
    Rectangle (151,112 48x32), "CH3", colour toggle: g_xHMI_EL2904Ch3
    Rectangle (203,112 48x32), "CH4", colour toggle: g_xHMI_EL2904Ch4
    Label (153,58 99x23), "EL2904 Outputs"
    Button (29,226 107x52), "Safety Group Err Ack"
        OnMouseDown: execute { g_xHMI_ErrAckPB := TRUE ; }
        OnMouseUp: execute { g_xHMI_ErrAckPB := FALSE ; }
    Button (148,226 107x52), "EStop Reset"
        OnMouseDown: execute { g_xHMI_EStopResetPB := TRUE ; }
        OnMouseUp: execute { g_xHMI_EStopResetPB := FALSE ; }
    Rectangle (30,153 226x32), "Safety Group1 Com Error", colour toggle: g_xHMI_SafetyGroup1_COMerrorLT
    Rectangle (29,189 226x32), "Safety Group1 FB Error", colour toggle: g_xHMI_SafetyGroup1_FBerrorLT
    Label (50,283 133x26), "Safety I/O Errors"
    Button (28,543 83x42), "EtherCAT Diag1"
        OnMouseClick: change screen: EtherCAT_Diag1
    Button (116,543 83x42), "EtherCAT Diag2"
        OnMouseClick: change screen: EtherCAT_Diag2
    Button (29,588 169x42), "TwinCAT INFO"
        OnMouseClick: change screen: TwinCAT_INFO
    RoundedRectangle (262,81 453x52)
    Label (449,80 224x26), "Safety Group INFO"
    Label (267,89 135x26), "Safety Group Status"
    RoundedRectangle (262,139 453x140)
    Label (449,137 224x26), "Safety Connection INFO"
    Label (267,146 203x26), "Connection 1 (EL1904)"
    Label (267,209 203x26), "Connection 2 (EL2904)"
    RoundedRectangle (202,285 513x360)
    Label (449,283 224x26), "Safety Function Block INFO"
    Label (268,313 50x26), "AND#1"
    Label (268,362 51x25), "EStop"
    Button (379,14 110x27), "AX5805"
        OnMouseClick: change screen: AX5805_Specific_Diagnostics
    Button (379,45 110x27), "EL6900"
        OnMouseClick: change screen: EL6900_Specific_Diagnostics
    Button (492,14 110x27), "EL1904"
        OnMouseClick: change screen: EL1904_Specific_Diagnostics
    Button (492,45 110x27), "EL6930"
        OnMouseClick: change screen: EL6930_Specific_Diagnostics
    Button (605,14 110x27), "EP1908"
        OnMouseClick: change screen: EP1908_Specific_Diagnostics
    Button (605,45 110x27), "EL2904"
        OnMouseClick: change screen: EL2904_Specific_Diagnostics
    Rectangle (267,107 321x22), "%s", text variable: g_sHMI_StatusGroup1
    Rectangle (267,163 321x22), "State: %s", text variable: g_sHMI_StateConn1
    Rectangle (267,178 386x22), "Diagnostic: %s", text variable: g_sHMI_DiagConn1
    Rectangle (267,226 321x22), "State: %s", text variable: g_sHMI_StateConn2
    Rectangle (267,242 389x22), "Diagnostic: %s", text variable: g_sHMI_DiagConn2
    Rectangle (268,331 439x22), "State: %s", text variable: g_sHMI_StatusAND1
    Rectangle (268,378 439x22), "State: %s", text variable: g_sHMI_StatusEStop1
    Rectangle (268,393 439x22), "Diagnostic: %s", text variable: g_sHMI_DiagEStop1
    Rectangle (268,439 439x22), "State: %s", text variable: g_sHMI_StatusAND2
    Label (268,421 54x26), "AND#2"
    Rectangle (268,488 439x22), "State: %s", text variable: g_sHMI_StatusTON
    Label (268,471 36x26), "TON"
    Rectangle (268,535 439x22), "State: %s", text variable: g_sHMI_StatusTOF
    Label (268,518 33x26), "TOF"
    Label (268,571 34x18), "EDM"
    Rectangle (268,584 439x22), "State: %s", text variable: g_sHMI_StatusEDM
    Rectangle (268,600 439x22), "Diagnostic: %s", text variable: g_sHMI_DiagEDM
    Rectangle (207,377 60x30), "EStop FB Error", colour toggle: g_xHMI_EStop_errorLT
    Rectangle (207,425 60x30), "EStop Complete", colour toggle: g_xHMI_EStop_CompleteLT
    Rectangle (207,475 60x30), "TON Complete", colour toggle: g_xHMI_EStop_ON_Delay_CompleteLT
    Rectangle (207,524 60x30), "TOF Complete", colour toggle: g_xHMI_EStop_OFF_Delay_CompleteLT
    Rectangle (207,584 60x30), "EDM FB Error", colour toggle: g_xHMI_EDMerrorLT
    Group (45,308 141x30)
        Button (0,0 141x30), colour toggle: g_xHMI_EL6900_General_Error
            OnMouseClick: change screen: AX5805_Specific_Diagnostics
            OnMouseUp: execute { g_xHMI_ErrAckPB := FALSE ; }
        Label (10,3 121x25), "EL6900 Error", invisible if: NOT g_xHMI_EL6900_General_Error
        Label (10,3 121x25), "EL6900 OK", invisible if: g_xHMI_EL6900_General_Error
    Group (45,345 141x30)
        Button (0,0 141x30), colour toggle: g_xHMI_EL6930_General_Error
            OnMouseClick: change screen: AX5805_Specific_Diagnostics
            OnMouseUp: execute { g_xHMI_ErrAckPB := FALSE ; }
        Label (10,3 121x25), "EL6930 Error", invisible if: NOT g_xHMI_EL6930_General_Error
        Label (10,3 121x25), "EL6930 OK", invisible if: g_xHMI_EL6930_General_Error
    Group (45,382 141x30)
        Button (0,0 141x30), colour toggle: g_xHMI_EL1904_General_Error
            OnMouseClick: change screen: AX5805_Specific_Diagnostics
            OnMouseUp: execute { g_xHMI_ErrAckPB := FALSE ; }
        Label (10,3 121x25), "EL1904 Error", invisible if: NOT g_xHMI_EL1904_General_Error
        Label (10,3 121x25), "EL1904 OK", invisible if: g_xHMI_EL1904_General_Error
    Group (44,419 141x30)
        Button (0,0 141x30), colour toggle: g_xHMI_EP1908_General_Error
            OnMouseClick: change screen: AX5805_Specific_Diagnostics
            OnMouseUp: execute { g_xHMI_ErrAckPB := FALSE ; }
        Label (10,3 121x25), "EP1908 Error", invisible if: NOT g_xHMI_EP1908_General_Error
        Label (10,3 121x25), "EP1908 OK", invisible if: g_xHMI_EP1908_General_Error
    Group (45,455 141x30)
        Button (0,0 141x30), colour toggle: g_xHMI_EL2904_General_Error
            OnMouseClick: change screen: AX5805_Specific_Diagnostics
            OnMouseUp: execute { g_xHMI_ErrAckPB := FALSE ; }
        Label (10,3 121x25), "EL2904 Error", invisible if: NOT g_xHMI_EL2904_General_Error
        Label (10,3 121x25), "EL2904 OK", invisible if: g_xHMI_EL2904_General_Error
    Group (45,491 141x30)
        Button (0,0 141x30), colour toggle: g_xHMI_AX5805_General_Error
            OnMouseClick: change screen: AX5805_Specific_Diagnostics
            OnMouseUp: execute { g_xHMI_ErrAckPB := FALSE ; }
        Label (10,3 121x25), "AX5805 Error", invisible if: NOT g_xHMI_AX5805_General_Error
        Label (10,3 121x25), "AX5805 OK", invisible if: g_xHMI_AX5805_General_Error
END_VISUALIZATION

// ---- VISUs/TwinSAFE.TcVIS
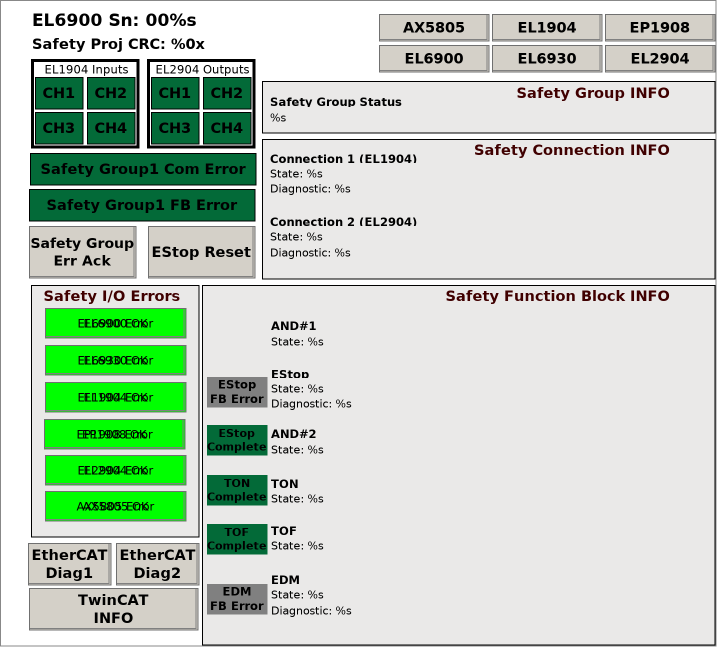
VISUALIZATION TwinSAFE  // 717x647
    RoundedRectangle (31,285 168x252)
    Rectangle (31,59 108x89)
    Rectangle (29,9 219x22), "EL6900 Sn: 00%s", text variable: g_udiHMI_SerialNumber
    Rectangle (29,33 232x22), "Safety Proj CRC: %0x", text variable: g_uiHMI_ProjectCRC
    Rectangle (35,77 48x32), "CH1", colour toggle: g_xHMI_EL1904Ch1
    Rectangle (87,77 48x32), "CH2", colour toggle: g_xHMI_EL1904Ch2
    Rectangle (35,112 48x32), "CH3", colour toggle: g_xHMI_EL1904Ch3
    Rectangle (87,112 48x32), "CH4", colour toggle: g_xHMI_EL1904Ch4
    Label (37,58 99x23), "EL1904 Inputs"
    Rectangle (147,59 108x89)
    Rectangle (151,77 48x32), "CH1", colour toggle: g_xHMI_EL2904Ch1
    Rectangle (203,77 48x32), "CH2", colour toggle: g_xHMI_EL2904Ch2
    Rectangle (151,112 48x32), "CH3", colour toggle: g_xHMI_EL2904Ch3
    Rectangle (203,112 48x32), "CH4", colour toggle: g_xHMI_EL2904Ch4
    Label (153,58 99x23), "EL2904 Outputs"
    Button (29,226 107x52), "Safety Group Err Ack"
        OnMouseDown: execute { g_xHMI_ErrAckPB := TRUE ; }
        OnMouseUp: execute { g_xHMI_ErrAckPB := FALSE ; }
    Button (148,226 107x52), "EStop Reset"
        OnMouseDown: execute { g_xHMI_EStopResetPB := TRUE ; }
        OnMouseUp: execute { g_xHMI_EStopResetPB := FALSE ; }
    Rectangle (30,153 226x32), "Safety Group1 Com Error", colour toggle: g_xHMI_SafetyGroup1_COMerrorLT
    Rectangle (29,189 226x32), "Safety Group1 FB Error", colour toggle: g_xHMI_SafetyGroup1_FBerrorLT
    Label (50,283 133x26), "Safety I/O Errors"
    Button (28,543 83x42), "EtherCAT Diag1"
        OnMouseClick: change screen: EtherCAT_Diag1
    Button (116,543 83x42), "EtherCAT Diag2"
        OnMouseClick: change screen: EtherCAT_Diag2
    Button (29,588 169x42), "TwinCAT INFO"
        OnMouseClick: change screen: TwinCAT_INFO
    RoundedRectangle (262,81 453x52)
    Label (449,80 224x26), "Safety Group INFO"
    Label (267,89 135x26), "Safety Group Status"
    RoundedRectangle (262,139 453x140)
    Label (449,137 224x26), "Safety Connection INFO"
    Label (267,146 203x26), "Connection 1 (EL1904)"
    Label (267,209 203x26), "Connection 2 (EL2904)"
    RoundedRectangle (202,285 513x360)
    Label (449,283 224x26), "Safety Function Block INFO"
    Label (268,313 50x26), "AND#1"
    Label (268,362 51x25), "EStop"
    Button (379,14 110x27), "AX5805"
        OnMouseClick: change screen: AX5805_Specific_Diagnostics
    Button (379,45 110x27), "EL6900"
        OnMouseClick: change screen: EL6900_Specific_Diagnostics
    Button (492,14 110x27), "EL1904"
        OnMouseClick: change screen: EL1904_Specific_Diagnostics
    Button (492,45 110x27), "EL6930"
        OnMouseClick: change screen: EL6930_Specific_Diagnostics
    Button (605,14 110x27), "EP1908"
        OnMouseClick: change screen: EP1908_Specific_Diagnostics
    Button (605,45 110x27), "EL2904"
        OnMouseClick: change screen: EL2904_Specific_Diagnostics
    Rectangle (267,107 321x22), "%s", text variable: g_sHMI_StatusGroup1
    Rectangle (267,163 321x22), "State: %s", text variable: g_sHMI_StateConn1
    Rectangle (267,178 386x22), "Diagnostic: %s", text variable: g_sHMI_DiagConn1
    Rectangle (267,226 321x22), "State: %s", text variable: g_sHMI_StateConn2
    Rectangle (267,242 389x22), "Diagnostic: %s", text variable: g_sHMI_DiagConn2
    Rectangle (268,331 439x22), "State: %s", text variable: g_sHMI_StatusAND1
    Rectangle (268,378 439x22), "State: %s", text variable: g_sHMI_StatusEStop1
    Rectangle (268,393 439x22), "Diagnostic: %s", text variable: g_sHMI_DiagEStop1
    Rectangle (268,439 439x22), "State: %s", text variable: g_sHMI_StatusAND2
    Label (268,421 54x26), "AND#2"
    Rectangle (268,488 439x22), "State: %s", text variable: g_sHMI_StatusTON
    Label (268,471 36x26), "TON"
    Rectangle (268,535 439x22), "State: %s", text variable: g_sHMI_StatusTOF
    Label (268,518 33x26), "TOF"
    Label (268,571 34x18), "EDM"
    Rectangle (268,584 439x22), "State: %s", text variable: g_sHMI_StatusEDM
    Rectangle (268,600 439x22), "Diagnostic: %s", text variable: g_sHMI_DiagEDM
    Rectangle (207,377 60x30), "EStop FB Error", colour toggle: g_xHMI_EStop_errorLT
    Rectangle (207,425 60x30), "EStop Complete", colour toggle: g_xHMI_EStop_CompleteLT
    Rectangle (207,475 60x30), "TON Complete", colour toggle: g_xHMI_EStop_ON_Delay_CompleteLT
    Rectangle (207,524 60x30), "TOF Complete", colour toggle: g_xHMI_EStop_OFF_Delay_CompleteLT
    Rectangle (207,584 60x30), "EDM FB Error", colour toggle: g_xHMI_EDMerrorLT
    Group (45,308 141x30)
        Button (0,0 141x30), colour toggle: g_xHMI_EL6900_General_Error
            OnMouseClick: change screen: AX5805_Specific_Diagnostics
            OnMouseUp: execute { g_xHMI_ErrAckPB := FALSE ; }
        Label (10,3 121x25), "EL6900 Error", invisible if: NOT g_xHMI_EL6900_General_Error
        Label (10,3 121x25), "EL6900 OK", invisible if: g_xHMI_EL6900_General_Error
    Group (45,345 141x30)
        Button (0,0 141x30), colour toggle: g_xHMI_EL6930_General_Error
            OnMouseClick: change screen: AX5805_Specific_Diagnostics
            OnMouseUp: execute { g_xHMI_ErrAckPB := FALSE ; }
        Label (10,3 121x25), "EL6930 Error", invisible if: NOT g_xHMI_EL6930_General_Error
        Label (10,3 121x25), "EL6930 OK", invisible if: g_xHMI_EL6930_General_Error
    Group (45,382 141x30)
        Button (0,0 141x30), colour toggle: g_xHMI_EL1904_General_Error
            OnMouseClick: change screen: AX5805_Specific_Diagnostics
            OnMouseUp: execute { g_xHMI_ErrAckPB := FALSE ; }
        Label (10,3 121x25), "EL1904 Error", invisible if: NOT g_xHMI_EL1904_General_Error
        Label (10,3 121x25), "EL1904 OK", invisible if: g_xHMI_EL1904_General_Error
    Group (44,419 141x30)
        Button (0,0 141x30), colour toggle: g_xHMI_EP1908_General_Error
            OnMouseClick: change screen: AX5805_Specific_Diagnostics
            OnMouseUp: execute { g_xHMI_ErrAckPB := FALSE ; }
        Label (10,3 121x25), "EP1908 Error", invisible if: NOT g_xHMI_EP1908_General_Error
        Label (10,3 121x25), "EP1908 OK", invisible if: g_xHMI_EP1908_General_Error
    Group (45,455 141x30)
        Button (0,0 141x30), colour toggle: g_xHMI_EL2904_General_Error
            OnMouseClick: change screen: AX5805_Specific_Diagnostics
            OnMouseUp: execute { g_xHMI_ErrAckPB := FALSE ; }
        Label (10,3 121x25), "EL2904 Error", invisible if: NOT g_xHMI_EL2904_General_Error
        Label (10,3 121x25), "EL2904 OK", invisible if: g_xHMI_EL2904_General_Error
    Group (45,491 141x30)
        Button (0,0 141x30), colour toggle: g_xHMI_AX5805_General_Error
            OnMouseClick: change screen: AX5805_Specific_Diagnostics
            OnMouseUp: execute { g_xHMI_ErrAckPB := FALSE ; }
        Label (10,3 121x25), "AX5805 Error", invisible if: NOT g_xHMI_AX5805_General_Error
        Label (10,3 121x25), "AX5805 OK", invisible if: g_xHMI_AX5805_General_Error
END_VISUALIZATION

// ---- VISUs/TwinSAFE.TcVIS
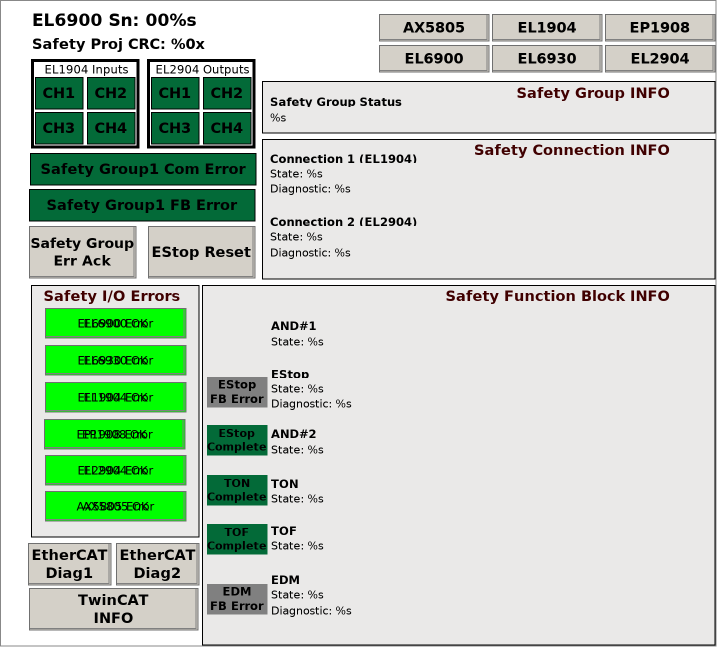
VISUALIZATION TwinSAFE  // 717x647
    RoundedRectangle (31,285 168x252)
    Rectangle (31,59 108x89)
    Rectangle (29,9 219x22), "EL6900 Sn: 00%s", text variable: g_udiHMI_SerialNumber
    Rectangle (29,33 232x22), "Safety Proj CRC: %0x", text variable: g_uiHMI_ProjectCRC
    Rectangle (35,77 48x32), "CH1", colour toggle: g_xHMI_EL1904Ch1
    Rectangle (87,77 48x32), "CH2", colour toggle: g_xHMI_EL1904Ch2
    Rectangle (35,112 48x32), "CH3", colour toggle: g_xHMI_EL1904Ch3
    Rectangle (87,112 48x32), "CH4", colour toggle: g_xHMI_EL1904Ch4
    Label (37,58 99x23), "EL1904 Inputs"
    Rectangle (147,59 108x89)
    Rectangle (151,77 48x32), "CH1", colour toggle: g_xHMI_EL2904Ch1
    Rectangle (203,77 48x32), "CH2", colour toggle: g_xHMI_EL2904Ch2
    Rectangle (151,112 48x32), "CH3", colour toggle: g_xHMI_EL2904Ch3
    Rectangle (203,112 48x32), "CH4", colour toggle: g_xHMI_EL2904Ch4
    Label (153,58 99x23), "EL2904 Outputs"
    Button (29,226 107x52), "Safety Group Err Ack"
        OnMouseDown: execute { g_xHMI_ErrAckPB := TRUE ; }
        OnMouseUp: execute { g_xHMI_ErrAckPB := FALSE ; }
    Button (148,226 107x52), "EStop Reset"
        OnMouseDown: execute { g_xHMI_EStopResetPB := TRUE ; }
        OnMouseUp: execute { g_xHMI_EStopResetPB := FALSE ; }
    Rectangle (30,153 226x32), "Safety Group1 Com Error", colour toggle: g_xHMI_SafetyGroup1_COMerrorLT
    Rectangle (29,189 226x32), "Safety Group1 FB Error", colour toggle: g_xHMI_SafetyGroup1_FBerrorLT
    Label (50,283 133x26), "Safety I/O Errors"
    Button (28,543 83x42), "EtherCAT Diag1"
        OnMouseClick: change screen: EtherCAT_Diag1
    Button (116,543 83x42), "EtherCAT Diag2"
        OnMouseClick: change screen: EtherCAT_Diag2
    Button (29,588 169x42), "TwinCAT INFO"
        OnMouseClick: change screen: TwinCAT_INFO
    RoundedRectangle (262,81 453x52)
    Label (449,80 224x26), "Safety Group INFO"
    Label (267,89 135x26), "Safety Group Status"
    RoundedRectangle (262,139 453x140)
    Label (449,137 224x26), "Safety Connection INFO"
    Label (267,146 203x26), "Connection 1 (EL1904)"
    Label (267,209 203x26), "Connection 2 (EL2904)"
    RoundedRectangle (202,285 513x360)
    Label (449,283 224x26), "Safety Function Block INFO"
    Label (268,313 50x26), "AND#1"
    Label (268,362 51x25), "EStop"
    Button (379,14 110x27), "AX5805"
        OnMouseClick: change screen: AX5805_Specific_Diagnostics
    Button (379,45 110x27), "EL6900"
        OnMouseClick: change screen: EL6900_Specific_Diagnostics
    Button (492,14 110x27), "EL1904"
        OnMouseClick: change screen: EL1904_Specific_Diagnostics
    Button (492,45 110x27), "EL6930"
        OnMouseClick: change screen: EL6930_Specific_Diagnostics
    Button (605,14 110x27), "EP1908"
        OnMouseClick: change screen: EP1908_Specific_Diagnostics
    Button (605,45 110x27), "EL2904"
        OnMouseClick: change screen: EL2904_Specific_Diagnostics
    Rectangle (267,107 321x22), "%s", text variable: g_sHMI_StatusGroup1
    Rectangle (267,163 321x22), "State: %s", text variable: g_sHMI_StateConn1
    Rectangle (267,178 386x22), "Diagnostic: %s", text variable: g_sHMI_DiagConn1
    Rectangle (267,226 321x22), "State: %s", text variable: g_sHMI_StateConn2
    Rectangle (267,242 389x22), "Diagnostic: %s", text variable: g_sHMI_DiagConn2
    Rectangle (268,331 439x22), "State: %s", text variable: g_sHMI_StatusAND1
    Rectangle (268,378 439x22), "State: %s", text variable: g_sHMI_StatusEStop1
    Rectangle (268,393 439x22), "Diagnostic: %s", text variable: g_sHMI_DiagEStop1
    Rectangle (268,439 439x22), "State: %s", text variable: g_sHMI_StatusAND2
    Label (268,421 54x26), "AND#2"
    Rectangle (268,488 439x22), "State: %s", text variable: g_sHMI_StatusTON
    Label (268,471 36x26), "TON"
    Rectangle (268,535 439x22), "State: %s", text variable: g_sHMI_StatusTOF
    Label (268,518 33x26), "TOF"
    Label (268,571 34x18), "EDM"
    Rectangle (268,584 439x22), "State: %s", text variable: g_sHMI_StatusEDM
    Rectangle (268,600 439x22), "Diagnostic: %s", text variable: g_sHMI_DiagEDM
    Rectangle (207,377 60x30), "EStop FB Error", colour toggle: g_xHMI_EStop_errorLT
    Rectangle (207,425 60x30), "EStop Complete", colour toggle: g_xHMI_EStop_CompleteLT
    Rectangle (207,475 60x30), "TON Complete", colour toggle: g_xHMI_EStop_ON_Delay_CompleteLT
    Rectangle (207,524 60x30), "TOF Complete", colour toggle: g_xHMI_EStop_OFF_Delay_CompleteLT
    Rectangle (207,584 60x30), "EDM FB Error", colour toggle: g_xHMI_EDMerrorLT
    Group (45,308 141x30)
        Button (0,0 141x30), colour toggle: g_xHMI_EL6900_General_Error
            OnMouseClick: change screen: AX5805_Specific_Diagnostics
            OnMouseUp: execute { g_xHMI_ErrAckPB := FALSE ; }
        Label (10,3 121x25), "EL6900 Error", invisible if: NOT g_xHMI_EL6900_General_Error
        Label (10,3 121x25), "EL6900 OK", invisible if: g_xHMI_EL6900_General_Error
    Group (45,345 141x30)
        Button (0,0 141x30), colour toggle: g_xHMI_EL6930_General_Error
            OnMouseClick: change screen: AX5805_Specific_Diagnostics
            OnMouseUp: execute { g_xHMI_ErrAckPB := FALSE ; }
        Label (10,3 121x25), "EL6930 Error", invisible if: NOT g_xHMI_EL6930_General_Error
        Label (10,3 121x25), "EL6930 OK", invisible if: g_xHMI_EL6930_General_Error
    Group (45,382 141x30)
        Button (0,0 141x30), colour toggle: g_xHMI_EL1904_General_Error
            OnMouseClick: change screen: AX5805_Specific_Diagnostics
            OnMouseUp: execute { g_xHMI_ErrAckPB := FALSE ; }
        Label (10,3 121x25), "EL1904 Error", invisible if: NOT g_xHMI_EL1904_General_Error
        Label (10,3 121x25), "EL1904 OK", invisible if: g_xHMI_EL1904_General_Error
    Group (44,419 141x30)
        Button (0,0 141x30), colour toggle: g_xHMI_EP1908_General_Error
            OnMouseClick: change screen: AX5805_Specific_Diagnostics
            OnMouseUp: execute { g_xHMI_ErrAckPB := FALSE ; }
        Label (10,3 121x25), "EP1908 Error", invisible if: NOT g_xHMI_EP1908_General_Error
        Label (10,3 121x25), "EP1908 OK", invisible if: g_xHMI_EP1908_General_Error
    Group (45,455 141x30)
        Button (0,0 141x30), colour toggle: g_xHMI_EL2904_General_Error
            OnMouseClick: change screen: AX5805_Specific_Diagnostics
            OnMouseUp: execute { g_xHMI_ErrAckPB := FALSE ; }
        Label (10,3 121x25), "EL2904 Error", invisible if: NOT g_xHMI_EL2904_General_Error
        Label (10,3 121x25), "EL2904 OK", invisible if: g_xHMI_EL2904_General_Error
    Group (45,491 141x30)
        Button (0,0 141x30), colour toggle: g_xHMI_AX5805_General_Error
            OnMouseClick: change screen: AX5805_Specific_Diagnostics
            OnMouseUp: execute { g_xHMI_ErrAckPB := FALSE ; }
        Label (10,3 121x25), "AX5805 Error", invisible if: NOT g_xHMI_AX5805_General_Error
        Label (10,3 121x25), "AX5805 OK", invisible if: g_xHMI_AX5805_General_Error
END_VISUALIZATION
